	IF TransportItemFound.ID <> '' THEN
		// Test the sorter item against the update item
		IF TransportItemFound.ID = TransportItemInSorter.ID THEN
			// Only update if it is different
			IF TransportItemFound.Destination <> TransportItemInSorter.Destination THEN
				IF .nSortBufferLogEnable.BUFFER_UPDATEDEST THEN
					sMessage := CONCAT(' Item: ', TransportItemInSorter.ID);
					sMessage := CONCAT(sMessage,' Index: ');
					sMessage := CONCAT(sMessage, UDINT_TO_STRING(TransportSorterIndex));
					sMessage := CONCAT(sMessage,' Orig Dest: ');
					sMessage := CONCAT(sMessage, DINT_TO_STRING(TransportItemInSorter.Destination));
					sMessage := CONCAT(sMessage,' Orig DeviceID ');
					sMessage := CONCAT(sMessage, TransportItemInSorter.DeviceID);
					// Write to the Error List
					ADSLOGSTR( msgCtrlMask := ADSLOG_MSGTYPE_HINT OR ADSLOG_MSGTYPE_LOG
						, msgFmtStr := 'Dest Updated After Induct: %s'
						, strArg := sMessage);
				END_IF
				// Update the Destination. If the destination is unavailable, it has been already been set to the default
				TransportItemInSorter.Destination := TransportItemFound.Destination;
				TransportItemInSorter.DeviceID := TransportItemFound.DeviceID;
				TransportItemInSorter.MessageType := TransportItemFound.MessageType;
				TransportItemInSorter.Status := TransportItemFound.Status;
				TransportItemInSorter.ExtStatus := TransportItemFound.ExtStatus;
	
				IF .nSortBufferLogEnable.BUFFER_UPDATEDEST THEN
					sMessage := CONCAT(' Item: ', TransportItemInSorter.ID);
					sMessage := CONCAT(sMessage,' Index: ');
					sMessage := CONCAT(sMessage, UDINT_TO_STRING(TransportSorterIndex));
					sMessage := CONCAT(sMessage,' New Dest: ');
					sMessage := CONCAT(sMessage, DINT_TO_STRING(TransportItemInSorter.Destination));
					sMessage := CONCAT(sMessage,' New DeviceID ');
					sMessage := CONCAT(sMessage, TransportItemInSorter.DeviceID);
					// Write to the Error List
					ADSLOGSTR( msgCtrlMask := ADSLOG_MSGTYPE_HINT OR ADSLOG_MSGTYPE_LOG
						, msgFmtStr := 'Dest Updated After Induct: %s'
						, strArg := sMessage);
				END_IF
			END_IF
			// Make sure that the destination update makes it to the item being inducted into the sorter
			IF st_UpdateItem.Item.ID <> '' THEN
				IF st_UpdateItem.Item.ID = TransportItemFound.ID THEN
					IF st_UpdateItem.Item.Destination <> TransportItemFound.Destination THEN
						IF .nSortBufferLogEnable.BUFFER_UPDATEDEST THEN
							// Log the original destination
							sMessage := CONCAT(' Item: ', st_UpdateItem.Item.ID);
							sMessage := CONCAT(sMessage, ' Pulses: ');
							sMessage := CONCAT(sMessage, UDINT_TO_STRING(st_Sorter.EncoderCounts));
							sMessage := CONCAT(sMessage,' Orig Dest: ');
							sMessage := CONCAT(sMessage, DINT_TO_STRING(st_UpdateItem.Item.Destination));
							// Write to the Error List
							ADSLOGSTR( msgCtrlMask := ADSLOG_MSGTYPE_HINT OR ADSLOG_MSGTYPE_LOG
								, msgFmtStr := 'Induct Dest Changed: %s'
								, strArg := sMessage);
						END_IF
						// Update the Destination
						st_UpdateItem.Item.Destination := TransportItemFound.Destination;
						// Log the new destination
						IF .nSortBufferLogEnable.BUFFER_UPDATEDEST THEN
							sMessage := CONCAT(' Item: ', st_UpdateItem.Item.ID);
							sMessage := CONCAT(sMessage, ' Pulses: ');
							sMessage := CONCAT(sMessage, UDINT_TO_STRING(st_Sorter.EncoderCounts));
							sMessage := CONCAT(sMessage,' New Dest: ');
							sMessage := CONCAT(sMessage, DINT_TO_STRING(st_UpdateItem.Item.Destination));
							// Write to the Error List
							ADSLOGSTR( msgCtrlMask := ADSLOG_MSGTYPE_HINT OR ADSLOG_MSGTYPE_LOG
								, msgFmtStr := 'Induct Dest Changed: %s'
								, strArg := sMessage);
						END_IF
					END_IF
				END_IF
			ELSE
				IF .nSortBufferLogEnable.BUFFER_UPDATEDEST THEN
					sMessage := CONCAT(' Item: ', TransportItemInSorter.ID);
					sMessage := CONCAT(sMessage,' Index: ');
					sMessage := CONCAT(sMessage, UDINT_TO_STRING(TransportSorterIndex));
					sMessage := CONCAT(sMessage,' Orig Dest: ');
					sMessage := CONCAT(sMessage, DINT_TO_STRING(TransportItemInSorter.Destination));
					// Write to the Error List
					ADSLOGSTR( msgCtrlMask := ADSLOG_MSGTYPE_HINT OR ADSLOG_MSGTYPE_LOG
						, msgFmtStr := 'Dest Received After Induct: %s'
						, strArg := sMessage);
				END_IF
				
			END_IF
		END_IF
	END_IF

	// Put the updated record back into the array
	aItems[TransportSorterIndex] := TransportItemInSorter;
	
//==================================================
// 	Done procesing Transport information
//
//	Begin processing Update/Exit information
//==================================================
	
	// For exits, start from the current encoder count and work forward
	ExitSorterIndex := F_CalculateIndex(Offset := UpdateIndexCounter
										, InitialValue := st_Sorter.EncoderCounts
										, BufferSize := ItemsArraySize);

	// Identify the Item we are testing
	ExitItemInSorter := aItems[ExitSorterIndex];

	// Populated ID identifies an item in the sorter
	// Between the two Divert status codes indicates that the item has attempted to divert
	IF ExitItemInSorter.ID <> '' THEN
		// Capture the Item encoder index and the Item at the current index
		//  This represents the first item record for this item
		//  It is captured to log the start index to allow this first record to be updated
		//  when the item is completely diverted
		IF ExitItemFound.Item.ID = '' THEN
			ExitItemFound.Counts := ExitSorterIndex;
			ExitItemFound.Item := ExitItemInSorter;
			IF ExitItemFound.Item.Status = E_StatusCode.Divert_Complete THEN
				ExitComplete := TRUE;
			END_IF
		END_IF
		// When ExitComplete is TRUE, and the ID's match, clear out this Item
		IF ExitComplete THEN
			IF ExitItemInSorter.ID = ExitItemFound.Item.ID THEN
				IF aItems[ExitSorterIndex].ID <> '' THEN
					IF .nSortBufferLogEnable.BUFFER_DUMP THEN
						sMessage := CONCAT(' Item: ', aItems[ExitSorterIndex].ID);
						sMessage := CONCAT(sMessage,' Index: ');
						sMessage := CONCAT(sMessage, UDINT_TO_STRING(ExitSorterIndex));
						sMessage := CONCAT(sMessage,' Item Status: ');
						sMessage := CONCAT(sMessage, DINT_TO_STRING(aItems[ExitSorterIndex].Status));
						sMessage := CONCAT(sMessage,' Item Ext Status: ');
						sMessage := CONCAT(sMessage, DINT_TO_STRING(aItems[ExitSorterIndex].ExtStatus));
						// Write to the Error List
						ADSLOGSTR( msgCtrlMask := ADSLOG_MSGTYPE_HINT OR ADSLOG_MSGTYPE_LOG
							, msgFmtStr := 'Exit Complete Dump Info: %s'
							, strArg := sMessage);
					END_IF
				END_IF
				aItems[ExitSorterIndex] := BlankItem;
			END_IF
		// When ExitComplete is FALSE, test for a diverting/diverted item
		ELSE
			// Detect when this item is in a diverting state
			IF (ExitItemInSorter.Status >= E_StatusCode.Diverting
			   OR ExitItemInSorter.Status <= E_StatusCode.Divert_Success)
			   THEN
			   	ExitInDivert := TRUE;
				(*
					Status value increase from Diverting to Divert_Complete
					Codes to indicate divert disposition are between Diverting and Divert_Detected
					Divert_Full and Diverting are set in FB_DivertDecision/FB_DivertControl
					Divert_Detected, Divert_Success, and Divert_Missed are set in FB_ConfirmCheck
				*)
				ExitDiverting := TRUE;
				IF ExitItemInSorter.Status = E_StatusCode.Divert_Detected THEN
					ExitDetected := TRUE;
				END_IF
				// Once the divert is successful, we are no longer "diverting"
				IF ExitItemInSorter.Status = E_StatusCode.Divert_Success THEN
					ExitSuccess := TRUE;
					ExitDiverting := FALSE;
				END_IF
				(*	
					ExitItemInSorter is the current item being examined
					ExitItemFound.Item is a copy of the Array item at ExitItemFound.Counts
					ExitItemFound.Counts references the Array index of the first record associated with this item
					When a Status/ExtStatus of greater value is detected, the first record Status/ExtStatus is overwritten
					The ExitItemFound.Item.Status/.ExtStatus is also updated
				*)
				IF ExitItemInSorter.Status > aItems[ExitItemFound.Counts].Status THEN
					aItems[ExitItemFound.Counts].Status := ExitItemInSorter.Status;
					ExitItemFound.Item.Status := ExitItemInSorter.Status;
				END_IF
				IF ExitItemInSorter.ExtStatus > aItems[ExitItemFound.Counts].ExtStatus THEN
					aItems[ExitItemFound.Counts].ExtStatus := ExitItemInSorter.ExtStatus;
					ExitItemFound.Item.ExtStatus := ExitItemInSorter.ExtStatus;
				END_IF
			END_IF
			aItems[ExitSorterIndex].Status := ExitItemFound.Item.Status;
		END_IF
	ELSE
		(*
			This path is followed when the ExitItemInSorter.ID is empty, which indicates
			that the array record associated with this index is not occupied

			ExitInDivert, ExitDiverting and ExitSuccess are all set while the .ID is not empty
		*)
		// This item was in a "diverting" state
		IF ExitInDivert THEN
			// This item is not currently diverting
			IF NOT ExitDiverting THEN
				// Only change to a Divert_Success if a Divert_Success was detected
				// Any other status is captured in the ELSE clause of the CASE statement
				IF ExitSuccess THEN
					ExitItemFound.Item.Status := E_StatusCode.Divert_Success;
				END_IF
				ExitItemFound.Item.CapturedInMetrics := TRUE;
				ExitItemFound.Item.MessageType := E_MessageIds.TransportComplete_26;
				fb_UpdateBuffer.AddItem(ExitItemFound.Item);
				aItems[ExitItemFound.Counts].Status := E_StatusCode.Divert_Complete;
			END_IF
		END_IF
		// Clear the last detected Exit item
		ExitItemFound.Item := BlankItem;
		// Reset the Detection booleans
		ExitInDivert := FALSE;
		ExitDiverting := FALSE;
		ExitDetected := FALSE;
		ExitSuccess := FALSE;
		ExitComplete := FALSE;
	END_IF
END_FOR

// If the ID is populated, we didn't find a match to update
IF st_ToUpdate.Item.ID <> '' THEN
	IF .nSortBufferLogEnable.BUFFER_UNASSIGNED THEN
		sMessage := CONCAT(' Item: ', st_ToUpdate.Item.ID);
		// Write to the Error List
		ADSLOGSTR( msgCtrlMask := ADSLOG_MSGTYPE_HINT OR ADSLOG_MSGTYPE_LOG
			, msgFmtStr := 'Item Not Updated: %s'
			, strArg := sMessage);
	END_IF
	st_ToUpdate.Item.Status := E_StatusCode.Assign_NotFound;
	st_ToUpdate.Item.DeviceID := st_Sorter.Config.Name;
	st_ToUpdate.Item.MessageType := E_MessageIds.TransportResponse_25;
	fb_UpDateBuffer.AddItem(st_ItemToAdd := st_ToUpdate.Item);
	st_ToUpdate.Item := BlankItem;
END_IF

END_PROGRAM

// ---- POUs/FunctionBlocks/Sorter/SorterExample.TcPOU
PROGRAM SorterExample
VAR
	nSorterClearIdx				: DINT;
	bSimulate					: BOOL := FALSE;	// Indicates when runing a simulation
	BlankItem					: ST_Item := (ID := ''
												, UniqueID := 0
												, Destination := 0
												, Status := E_StatusCode.No_Status
												, ExtStatus := E_StatusCode.No_Status
												, DeviceID := ''
												, MessageType := E_MessageIds.NoMessage_00);
	
	st_ToInduct					: ST_ItemTemporary;	// This is the next item to be inducted onto the sorter
	st_Inducting				: ST_ItemTemporary;	// This is the next item to be inducted onto the sorter
	st_InductUpdate				: ST_ItemTemporary;	// This is to update an item already being inducted
	{attribute 'OPC.UA.DA' := '1'}
	st_Sorter					: ST_Sorter;
	{attribute 'OPC.UA.DA' := '1'}
	aSorterDiverts 				: ARRAY[DIVERTMIN..NUMBEROFDIVERTS] OF ST_Divert;

	st_SorterEncoder 			: ST_Encoder;
	fb_SorterEncoder 			: FB_ProcessEncoder;
	{attribute 'OPC.UA.DA' := '1'}
	ENC_Raw	AT %I*:	UINT;	// Raw Encoder Value
	tEncoderOK			: TON;
	nLastEncoderCount	: UDINT;

	{attribute 'OPC.UA.DA' := '1'}
	fb_SortMetrics				: FB_Metrics;

	In_DefaultDestination AT %I*	: DINT;	// Input default destination update from Host messaging(MsgControl.RECEIVE)

	fb_CommissionSorterDiverts	: FB_DivertCommission;
	rInductPE					: R_TRIG; 	// Capture the Rising edge of the Induct PE
	fInductPE					: F_TRIG; 	// Capture the Falling edge of the Induct PE

	rDischargePE				: R_TRIG; 	// Capture the Rising edge of the Discharge PE
	fDischargePE				: F_TRIG; 	// Capture the Falling edge of the Discharge PE

	st_TempItem					: ST_ItemTemporary;	// Store temporary Item info until BCR data is received

	DivertToCommission			: UINT := 0;	// Non-zero value will send all items to this divert

	sMessage			: STRING;

	ClearSorterArray	: BOOL;

	FB_DivertLog		: FB_DivertLog;
	
	SorterDischargeItem	: ST_Item;

END_VAR

VAR PERSISTENT
	aSorterItems 				: ARRAY[SORTERENCODERMIN..SORTERENCODERMAX] OF ST_Item;	// Persist the Items to Sort array
	{attribute 'OPC.UA.DA' := '1'}
	st_SorterCfg				: ST_SorterConfig; 	// Persist Sorter configuration
	{attribute 'OPC.UA.DA' := '1'}
	aSorterDivertsCfgs 			: ARRAY[DIVERTMIN..NUMBEROFDIVERTS] OF ST_DivertCfg; 	// Persist Sorter Configuration
END_VAR

VAR CONSTANT
	SORTERMASKSIZE				: UINT := 11;		// Number of bits to mask into the Encoder Count, will define the size of the SORTERENCODERMAX value
	{attribute 'OPC.UA.DA' := '1'}
	NUMBEROFDIVERTS				: DINT := 3;
	DIVERTMIN					: DINT := 1;
	{attribute 'OPC.UA.DA' := '1'}
	SORTERENCODERMAX			: UDINT := ((LREAL_TO_UDINT(EXPT(2,SORTERMASKSIZE)))-1); // Calculated size based on the bitmask 
	{attribute 'OPC.UA.DA' := '1'}
	SORTERENCODERMIN			: UDINT := 0;

END_VAR

// Sorter clear when the system is restarted or downloaded (INIT=TRUE for first scan)
IF (GVL_IO.INIT AND NOT st_SorterCfg.RetainOnRestart) OR ClearSorterArray THEN
	FOR nSorterClearIdx := UDINT_TO_DINT(SORTERENCODERMIN) TO UDINT_TO_DINT(SORTERENCODERMAX) BY 1 DO
		IF nSorterLogEnable.SORTER_DUMP THEN
			IF aSorterItems[nSorterClearIdx].ID <> '' THEN
				IF .nSorterLogEnable.SORTER_DUMP THEN
					sMessage := CONCAT(' Item: ', aSorterItems[nSorterClearIdx].ID);
					sMessage := CONCAT(sMessage,' Index: ');
					sMessage := CONCAT(sMessage, DINT_TO_STRING(nSorterClearIdx));
					// Write to the Error List
					ADSLOGSTR( msgCtrlMask := ADSLOG_MSGTYPE_HINT OR ADSLOG_MSGTYPE_LOG
						, msgFmtStr := 'Array Dump Info: %s'
						, strArg := sMessage);
				END_IF
			END_IF
		END_IF
		aSorterItems[nSorterClearIdx] := BlankItem;
	END_FOR
	ClearSorterArray := FALSE;
END_IF

// Setup and process the Sorter Encoder
st_SorterEncoder.EncoderRawCount := ENC_Raw;
st_SorterEncoder.BitMaskSize := SORTERMASKSIZE;
fb_SorterEncoder(Encoder := st_SorterEncoder, Simulate := bSimulate);

(*
	Initializes the Diverts.  
*)
{warning 'TODO: Fix references to Full and Confirm PE'}
{warning 'TODO: Add Configuration for all Diverts'}
aSorterDiverts[1].Config := aSorterDivertsCfgs[1];
aSorterDiverts[1].FullPE := TRUE;
aSorterDiverts[1].ConfirmPE := TRUE;

fb_CommissionSorterDiverts(
			//InductTrigger := Photoeyes.PE_22441.Out,
			ReferenceValue := st_SorterEncoder.CurrentCount, 
			//DischargeTrigger := Photoeyes.PE_23121.Out_OffFltrd,
			TestTime := T#10S, Diverts := aSorterDiverts);

// Provide a "hard-coded" default destination.
IF st_SorterCfg.DefaultDestination <= 0 THEN
	st_SorterCfg.DefaultDestination := 1;
END_IF						

// Name of the sorter equipment
//st_SorterCfg.Name := Conveyors.cfgP8005Label;
st_SorterCfg.DivertCount := NUMBEROFDIVERTS;
IF DivertToCommission > 0 THEN
	st_SorterCfg.DefaultDestination := DivertToCommission;
END_IF
st_Sorter.EncoderCounts := st_SorterEncoder.CurrentCount;
//st_Sorter.InductPE := PhotoEyes.PE_22441.Out_OnFltrd;
//st_Sorter.DischargePE := Photoeyes.PE_23081.Out_OnFltrd;

// Test the Encoder
//tEncoderOK.IN := (Conveyors.P8005_VFD.IsRunning AND (st_Sorter.EncoderCounts = nLastEncoderCount));
tEncoderOK(PT:=T#1S);

// OK when Q is not on, but the alarm is reversed
//GVL_IO.ENC_11321_OK := tEncoderOK.Q;

// Publish the sorter name
//GVL_IO.SorterName := st_SorterCfg.Name;

// Sorter
(*
	ProcessBuffers processes all associated buffers (Sorter/Divert/Arrival/Transport/Update)
	Items arriving at the sorter are detected and processed in this function block then deliverd to the SorterProgram
	Items inducted into sorter produce TransportResponse messages in this function block
	Items diverted off the sorter produce TransportComplete messages in this function block
*)
ProcessBuffers(st_NextToInduct := st_ToInduct
				, st_TempInductItem := st_TempItem
				, st_UpdateItem := st_Inducting
				, st_Sorter := st_Sorter
				, aDiverts := aSorterDiverts
				, aItems := aSorterItems
				, DivertToCommission := DivertToCommission
				, ItemsArrayMax := SORTERENCODERMAX
				, ItemsArrayMin := SORTERENCODERMIN);

// Capture rising and falling edge Triggers of the configured Sorter PE (Induct/Discharge)
rInductPE(CLK:= st_Sorter.InductPE, Q =>);
fInductPE(CLK:= st_Sorter.InductPE, Q =>);
rDischargePE(CLK:= st_Sorter.DischargePE, Q =>);
fDischargePE(CLK:= st_Sorter.DischargePE, Q =>);

// Prepare a dummy record for items that arrive before BCR data is received
// On the rising edge of the Induct PE
IF rInductPE.Q THEN
	IF .nSorterLogEnable.SORTER_INDUCT_PE THEN
		// Write to the Error List
		ADSLOGSTR( msgCtrlMask := ADSLOG_MSGTYPE_HINT OR ADSLOG_MSGTYPE_LOG
			, msgFmtStr := 'Induct PE Blocked : %s'
			, strArg := BOOL_TO_STRING(st_Sorter.InductPE)); 
	END_IF
	// Test for a UniqueID, which indicates that a Barcode has been received
	IF st_ToInduct.Item.UniqueID = 0 THEN
		// Capture and create relevant info
		st_TempItem.Counts := st_Sorter.EncoderCounts;
		st_TempItem.Item.UniqueID :=  UDINT_TO_DINT(st_Sorter.EncoderCounts);
		st_TempItem.Item.ID :=  CONCAT('T-', UDINT_TO_STRING(st_Sorter.EncoderCounts));
		st_TempItem.Item.Destination := st_SorterCfg.DefaultDestination;
		st_TempItem.Item.Status := E_StatusCode.UnidentifiedItem;
		IF .nSorterLogEnable.SORTER_TEMPID THEN
			ADSLOGSTR( msgCtrlMask := ADSLOG_MSGTYPE_HINT OR ADSLOG_MSGTYPE_LOG
				, msgFmtStr := 'Temp ID Assigned : %s'
				, strArg := st_TempItem.Item.ID);
		END_IF
	END_IF	
END_IF

// Clear the dummy record when the PE clears
// Items can only be inducted when the BCR info is received before or while the induct PE is blocked
IF fInductPE.Q THEN
	IF .nSorterLogEnable.SORTER_INDUCT_PE THEN
		// Write to the Error List
		ADSLOGSTR( msgCtrlMask := ADSLOG_MSGTYPE_HINT OR ADSLOG_MSGTYPE_LOG
			, msgFmtStr := 'Induct PE Blocked : %s'
			, strArg := BOOL_TO_STRING(st_Sorter.InductPE));
	END_IF
	// Clear the record
	st_TempItem.Counts := 0;
	st_TempItem.Item :=  BlankItem;
END_IF

(*
	SorterProgram is a separate Program
	Config portion of the st_sorter is separate to allow it be be persistent.
*)
st_sorter.Config := st_sorterCfg;
SorterProgram(st_Sorter := st_Sorter
		, In_ItemToInduct := st_ToInduct.Item
		, In_InductingItem := st_Inducting.Item
		, aItems := aSorterItems
		, aDiverts := aSorterDiverts
		, st_tempItem := st_TempItem
		, ItemsArrayMax := SORTERENCODERMAX
		, ItemsArrayMin := SORTERENCODERMIN
		, DivertArrayMax := DIVERTMIN
		, DivertArrayMin := NUMBEROFDIVERTS
		, st_DischargeItem => SorterDischargeItem);

// Log the diverts
FB_DivertLog(DivertArray := aSorterDiverts,
				DivertLogEnable := .nDivertLogEnable,
				EncoderCounts := st_SorterEncoder.CurrentCount);

END_PROGRAM

// ---- POUs/FunctionBlocks/Sorter/Functions/FB_FindDestination.TcPOU
FUNCTION_BLOCK FB_FindDestination
VAR_IN_OUT
	RoundRobin		:	ST_RoundRobin;
	aDiverts		:	ARRAY[*] OF ST_Divert;
	DestinationID	:	DINT;
END_VAR
VAR_INPUT
	SorterLogEnable	:	UDINT;
END_VAR
VAR_OUTPUT
	DestinationIndex	:	DINT;
	DestinationState	:	DINT;
END_VAR
VAR
	DivertArrayMin		:	DINT;
	DivertArrayMax		:	DINT;
	Last_Enabled	:	UINT;
	IndexCheck		:	DINT;
	sMessage		:	STRING;
END_VAR

// Get the upper and lower bounds of the divert array
DivertArrayMin := LOWER_BOUND(aDiverts,1);
DivertArrayMax := UPPER_BOUND(aDiverts,1);

//When a response is received, find the designated Destination
IF DestinationID >= 0 THEN
	IF SorterLogEnable.SORTER_DESTINATION_LU THEN
		sMessage := CONCAT(' Destination: ', DINT_TO_STRING(DestinationID));
		// Write to the Error List
		ADSLOGSTR( msgCtrlMask := ADSLOG_MSGTYPE_HINT OR ADSLOG_MSGTYPE_LOG
			, msgFmtStr := 'Lookup: %s'
			, strArg := sMessage);
	END_IF
	// Check to see if the Destination is defined as a round-robin destination for this sorter
	IF DestinationID = RoundRobin.Destination THEN
		// Test to see if the last enabled round robin destinations are still enabled
		// If they are different, restart the round-robin assignment to accommodate differences 
		IF RoundRobin.Enabled = Last_Enabled THEN
			// Test to see if the round robin assignments have all been met
			// If they have, clear and start over
			IF RoundRobin.Available = RoundRobin.Sent THEN
				RoundRobin.Sent := 0;
			END_IF
		ELSE
			// Capture the new enabled round-robin destinations
			// Restart the round robin assignments
			Last_Enabled := RoundRobin.Enabled;
			RoundRobin.Sent := 0;
		END_IF
		FOR IndexCheck := 0 TO 15 DO
			IF (
			   ((RoundRobin.Enabled AND LREAL_TO_UINT(EXPT(2,IndexCheck))) > 0) 
			   AND ((RoundRobin.Available AND LREAL_TO_UINT(EXPT(2,IndexCheck))) > 0)
			   AND NOT ((RoundRobin.Sent AND LREAL_TO_UINT(EXPT(2,IndexCheck))) > 0))
			   THEN
				RoundRobin.Sent := LREAL_TO_UINT(EXPT(2,IndexCheck)) OR RoundRobin.Sent;
				IF RoundRobin.aDestinations[IndexCheck] >= DivertArrayMin
				   AND RoundRobin.aDestinations[IndexCheck] <= DivertArrayMax
				   THEN
					DestinationIndex := RoundRobin.aDestinations[IndexCheck];
					DestinationID := aDiverts[DestinationIndex].Config.Number;
				ELSE
					DestinationIndex := DivertArrayMax;
				END_IF
				DestinationState := 0;
				EXIT;
			END_IF
		END_FOR
		IF SorterLogEnable.SORTER_DESTINATION_LU THEN
			sMessage := DINT_TO_STRING(DestinationIndex);
			sMessage := CONCAT(' Dest ID: ', DINT_TO_STRING(DestinationID));
			// Write to the Error List
			ADSLOGSTR( msgCtrlMask := ADSLOG_MSGTYPE_HINT OR ADSLOG_MSGTYPE_LOG
				, msgFmtStr := 'RoundRobin Dest: %s'
				, strArg := sMessage);
		END_IF
	ELSE
		DestinationIndex := DivertArrayMax;
		FOR IndexCheck := DivertArrayMin TO DivertArrayMax  DO
			IF aDiverts[IndexCheck].Config.Number = DestinationID THEN
				DestinationIndex := IndexCheck;
				DestinationState := 0;
				EXIT;
			END_IF
		END_FOR
		IF SorterLogEnable.SORTER_DESTINATION_LU THEN
			sMessage := DINT_TO_STRING(DestinationIndex);
			sMessage := CONCAT(' Dest ID: ', DINT_TO_STRING(DestinationID));
			// Write to the Error List
			ADSLOGSTR( msgCtrlMask := ADSLOG_MSGTYPE_HINT OR ADSLOG_MSGTYPE_LOG
				, msgFmtStr := 'Lookup Dest: %s'
				, strArg := sMessage);
		END_IF
	END_IF
END_IF

END_FUNCTION_BLOCK

// ---- POUs/Sorter_P6040.TcPOU
PROGRAM Sorter_P6040

VAR_IN_OUT
	In_ItemToInduct					: ST_Item;
	In_InductingItem				: ST_Item;
	st_tempItem						: ST_ItemTemporary;	// Temporary record used when barcode not yet received
	st_Sorter						: ST_Sorter;
	aDiverts						: ARRAY[Sorter.DIVERTMIN..Sorter.NUMBEROFDIVERTS] OF ST_DIVERT;
	aItems 							: ARRAY[Sorter.SORTERENCODERMIN..Sorter.SORTERENCODERMAX] OF ST_Item;
END_VAR

VAR_INPUT
	ItemsArrayMax		: UDINT;
	ItemsArrayMin		: UDINT;
	DivertArrayMax		: DINT;
	DivertArrayMin		: DINT;
END_VAR

VAR_OUTPUT
	st_DischargeItem	:	ST_Item;
END_VAR
VAR
	// Sorter Diagnostics
	aSorterDiagLog		: ST_ItemLogBuffer;
	fbSorterDiagLog		: FB_ItemLogBuffer;

	//Logging Variables
	UpdateSorterLog : FB_UpdateLog;
	
	//Induct Variables
	testEncoderCount		: UDINT;
	exitEncoderCount		: UDINT;
	lastCompareCount		: UDINT;
	updatingEncoderCount	: UDINT;

	tailendcount		: DINT := 0;
	inductindex 		: DINT;
	
	//Divert Variables
	fb_DivertDecision 		: FB_DivertDecision;
	fb_DivertFullMonitor  	: FB_DivertFullMonitor;
	DivertIndex				: DINT;
	Divertoffset			: INT;
	nTestItemIndex			: UDINT;
	Output2ItemIndex		: UDINT;

	// Confirm Check variables
	fb_ConfirmCheck 		: ARRAY[Sorter.DIVERTMIN..Sorter.NUMBEROFDIVERTS] OF FB_ConfirmCheck;
	st_ConfirmItem 			: ARRAY[Sorter.DIVERTMIN..Sorter.NUMBEROFDIVERTS] OF ST_Item;
	nConfirmItemIndex 		: UDINT;
	
	workingItem			: ST_Item;	// Actual item to induct

	LastItemInducted 	: STRING;
	nIndexToClear		: UDINT;	// Clear Item Array at this index
	nItemArraySize		: UDINT;

	rInductPE			: R_TRIG; 	// Capture the Rising edge of the Induct PE
	fInductPE			: F_TRIG; 	// Capture the Falling edge of the Induct PE
	sMessage			: STRING;

	st_DisplayItem		:st_Item;
	
	LogSorterDump: BOOL := FALSE;
END_VAR

// Initialize FB_ItemExtBuffer
fbSorterDiagLog(st_BufferData := aSorterDiagLog);

(*
// Test visu variables	
inductPE := SorterInductPE;
ItemsOut := Items;
ArrivalOut := ArrivalBuffer;
// End test variables
*)
(*
	Capture the Upper/Lower bound of relevant IO_OUT arrays for looping purposes
	ItemsArrayMax/Min for the sorter array slot count
*)
// Size is Max - Min + 1 to capture both extremes
nItemArraySize := ItemsArrayMax - ItemsArrayMin + 1;

FOR divertIndex := DivertArrayMin TO DivertArrayMax DO
	fb_DivertFullMonitor(Divert := aDiverts[divertIndex]);
END_FOR

(*
	Detect barcode receipt after item is already in Item array
	the tempItem is reset when the induct PE is cleared
	The tempItem is populated when the induct PE is blocked and there
	is not an associated barcode waiting to be inducted
*)
IF st_tempItem.Item.ID <> '' THEN
	// Test the IN_ItemToInduct.ID for a value
	// This record will be cleared as soon as it reaches the sorter loop
	IF In_ItemToInduct.ID <> '' THEN
		// The tempItem is overwritten with the IN_ItemToInduct after it is updated
		// But the starting encoder count is not changed so the same items can be updated
		// if the destination update is received while the item is still being inducted
		IF In_ItemToInduct.ID <> st_tempItem.Item.ID THEN 
			// Set the starting count for the testing/updating process
			// The testEncodeCount is incremented upon start, so we start -1 of the encoder count for the item
			testEncoderCount := f_CalculateIndex(Offset := -1, InitialValue:= st_tempItem.Counts, BufferSize := nItemArraySize);
			// Clear the length and start over
			In_ItemToInduct.Length := 0;
			st_tempItem.Item := In_ItemToInduct;
		END_IF 
		// Test for a change of destination after the barcode data has been received
		IF In_ItemToInduct.Destination <> st_tempItem.Item.Destination THEN 
			// Set the starting count for the testing/updating process
			// The testEncodeCount is incremented upon start, so we start -1 of the encoder count for the item
			testEncoderCount := f_CalculateIndex(Offset := -1, InitialValue:= st_tempItem.Counts, BufferSize := nItemArraySize);
			// Clear the length and start over
			In_ItemToInduct.Length := 0;
			// Copy the IN_ItemToInduct to prevent running this until something else in the record changes
			st_tempItem.Item := IN_ItemToInduct;
		END_IF
	END_IF 
END_IF


// Test for the rising edge of the induct PE
// Use this rising edge to log the IN_ItemToInduct record
rInductPE(CLK:= st_Sorter.InductPE, Q =>);

IF rInductPE.Q THEN
	IF .nSorterLogEnable.SORTER_INDUCT THEN
		sMessage := CONCAT(' Item: ', In_ItemToInduct.ID);
		sMessage := CONCAT(sMessage, ' Pulses: ');
		sMessage := CONCAT(sMessage, UDINT_TO_STRING(st_Sorter.EncoderCounts));
		// Write to the Error List
		ADSLOGSTR( msgCtrlMask := ADSLOG_MSGTYPE_HINT OR ADSLOG_MSGTYPE_LOG
			, msgFmtStr := 'Induct Info: %s'
			, strArg := sMessage);
	END_IF
END_IF
// Test for the falling edge of the induct PE
// Use this falling edge to clear the IN_ItemToInduct record
fInductPE(CLK:= st_Sorter.InductPE, Q =>);

IF fInductPE.Q THEN
	IF .nSorterLogEnable.SORTER_INDUCT THEN
		sMessage := CONCAT(' Item: ', In_ItemToInduct.ID);
		sMessage := CONCAT(sMessage,' Pulses: ');
		sMessage := CONCAT(sMEssage, UDINT_TO_STRING(st_Sorter.EncoderCounts));
		// Write to the Error List
		ADSLOGSTR( msgCtrlMask := ADSLOG_MSGTYPE_HINT OR ADSLOG_MSGTYPE_LOG
			, msgFmtStr := 'Cleared Induct Info: %s'
			, strArg := sMessage);
	END_IF
	// Clear the record
	In_InductingItem :=  BlankItem;
END_IF

// Process every array index between the current index and the last processed index
WHILE st_Sorter.EncoderCounts <> testEncoderCount DO

	// Capture the lastEncoderCount before changing it for comparison of last inducted items
	lastCompareCount := testEncoderCount;

	// Increment the testEncoderCount
	// The testEncoderCount variable will be used throughout the processing to ensure
	//	that all array elements are processed
	testEncoderCount := f_CalculateIndex(Offset := 1, InitialValue:= testEncoderCount, BufferSize := nItemArraySize);
	IF st_Sorter.InductPE THEN
	  	IF (In_ItemToInduct.ID <> '') THEN
			In_InductingItem := In_ItemToInduct;
			In_ItemToInduct := BlankItem;
			IF .nSorterLogEnable.SORTER_INDUCT_PE THEN
				sMessage := CONCAT(' Item: ', In_InductingItem.ID);
				sMessage := CONCAT(sMessage,' Pulses: ');
				sMessage := CONCAT(sMessage, UDINT_TO_STRING(st_Sorter.EncoderCounts));
				sMessage := CONCAT(sMessage,' Dest: ');
				sMessage := CONCAT(sMessage, DINT_TO_STRING(In_InductingItem.Destination));
				// Write to the Error List
				ADSLOGSTR( msgCtrlMask := ADSLOG_MSGTYPE_HINT OR ADSLOG_MSGTYPE_LOG
					, msgFmtStr := 'Inducting Info: %s'
					, strArg := sMessage);
			END_IF
		END_IF
	  	IF (In_InductingItem.ID <> '') THEN
			LastItemInducted := In_InductingItem.ID;
			IF aItems[testEncoderCount].ID <> '' THEN
				IF aItems[testEncoderCount].Status >= E_StatusCode.Diverting AND aItems[testEncoderCount].Status <= E_StatusCode.Divert_UnknownError THEN
					aItems[testEncoderCount].Status := E_StatusCode.Divert_UnknownError;
				END_IF
				UpdateSorterLog(Status := aItems[testEncoderCount].Status, ItemID := aItems[testEncoderCount].UniqueID);
			END_IF
		
			// Set the Item status
			In_InductingItem.Status := E_StatusCode.In_Sorter;

			// Check for destination full on the first pass, then ignore it.
		IF In_InductingItem.Length = 0 THEN
				IF aDiverts[In_InductingItem.DestinationIdx].Full THEN
					IF st_Sorter.Config.RecircUsed THEN
						In_InductingItem.Destination := st_Sorter.Config.RecircDestination;
						In_InductingItem.DestinationIdx := st_Sorter.Config.RecircDestIdx;
						In_InductingItem.ExtStatus := E_StatusCode.Divert_Recirculated;
					ELSE
						In_InductingItem.Destination := st_Sorter.Config.DefaultDestination;
						In_InductingItem.DestinationIdx := st_Sorter.Config.DefaultDestIdx;
						In_InductingItem.ExtStatus := E_StatusCode.Divert_Full;
					END_IF
				END_IF
			END_IF 
			// Clear the extend counter
			tailendcount := 0;

			// Copy the ItemToInduct to the WorkingItem that will be inducted
			workingItem := In_InductingItem;
			// Increment the Length on the ItemToInduct record, then it will be added to the array
			//  and the length will increment
			In_InductingItem.Length := In_InductingItem.Length +  1;
			// Determined by UniqueID = 0
		ELSE //If the item makes it to the sorter, but is not identified, induct the item with tempItem.Item
			LastItemInducted := 'UNKNOWN';
			(*UpdateSorterLog(Status := E_StatusCode.UnidentifiedItem, ItemID := st_tempItem.Item.UniqueID);*)

			// Process this the first time
			IF st_tempItem.Item.Length = 0 THEN
				IF aDiverts[st_Sorter.Config.DefaultDestIdx].Full THEN
					IF st_Sorter.Config.RecircUsed THEN
						st_tempItem.Item.Destination := st_Sorter.Config.RecircDestination;
						st_tempItem.Item.DestinationIdx := st_Sorter.Config.RecircDestIdx;
						st_tempItem.Item.ExtStatus := E_StatusCode.Divert_Recirculated;
					ELSE
						st_tempItem.Item.Destination := st_Sorter.Config.DefaultDestination;
						st_tempItem.Item.DestinationIdx := st_Sorter.Config.DefaultDestIdx;
						st_tempItem.Item.ExtStatus := E_StatusCode.Divert_Full;
					END_IF
				ELSE
					st_tempItem.Item.Destination := st_Sorter.Config.DefaultDestination;
					st_tempItem.Item.DestinationIdx := st_Sorter.Config.DefaultDestIdx;
				END_IF		
			END_IF
			// Copy the tempItem.Item to the WorkingItem that will be inducted
			workingItem := st_tempItem.Item;
			// Increment the Length on the ItemToInduct record, then it will be added to the array
			//  and the length will increment
			st_tempItem.Item.Length := st_tempItem.Item.Length +  1;
		END_IF

		// Induct everything
		aItems[testEncoderCount] := workingItem;
		fbSorterDiagLog.AddItem(workingItem);
	// Follow this path when the induct photo-eye is cleared
	ELSE
		// Extend the end of the item by a set amount, or to a mimimum length
		// Test to verify that the Item index is clear, and we are still extending the length of the item
		IF aItems[lastCompareCount].ID <> '' THEN
			IF tailendcount < st_Sorter.Config.TailEndLength AND st_Sorter.Config.TailEndLength > 0 THEN
				aItems[testEncoderCount] := aItems[lastCompareCount]; 
				fbSorterDiagLog.AddItem(aItems[lastCompareCount]);
				aItems[testEncoderCount].Length := aItems[testEncoderCount].Length + 1;
				tailendcount := tailendcount + 1;
			END_IF
			IF aItems[lastCompareCount].Length < st_Sorter.Config.MinimumLength AND st_Sorter.Config.MinimumLength > 0 THEN
				aItems[testEncoderCount] := aItems[lastCompareCount]; 
				fbSorterDiagLog.AddItem(aItems[lastCompareCount]);
				aItems[testEncoderCount].Length := aItems[testEncoderCount].Length + 1;
			END_IF
		END_IF
	END_IF
END_WHILE

// Process every array index between the current index and the last processed exit index
WHILE st_Sorter.EncoderCounts <> exitEncoderCount DO

	// Increment the exitEncoderCount
	// The exitEncoderCount variable will be used throughout the processing to ensure
	//	that all array elements are processed
	exitEncoderCount := f_CalculateIndex(Offset := 1, InitialValue:= exitEncoderCount, BufferSize := nItemArraySize);
	// Process the diverts relative to the current encoder count
	FOR divertIndex := DivertArrayMin TO DivertArrayMax DO
		// Get the distance to each divert, distance is the number of pulses to actuation
		Divertoffset := aDiverts[divertIndex].Config.Distance;
		// Calculate the index of the item to test for a divert
		// Subtract the offset from the current encoder count (exitEncoderCount)
		// As the encoder count increases, the current index pointer advances
		// Subtracting looks backwards into the sorter item array to test for items at the diverts
		//	distance that should be diverted
		nTestItemIndex := F_CalculateIndex(initialvalue := exitEncoderCount
										, offset := -(Divertoffset)
										, BufferSize := (ItemsArrayMax + 1));	
		//Setup Out2Item for energizing 2nd divert output
		Output2ItemIndex := F_CalculateIndex(initialvalue := exitEncoderCount
										, offset := -(Divertoffset + UINT_TO_INT(st_Sorter.Config.Output2Offset))
										, BufferSize := (ItemsArrayMax + 1));	
		// Log Diverts
		IF aItems[nTestItemIndex].DestinationIdx = divertIndex THEN
			IF .nSorterLogEnable.SORTER_DIVERTS THEN
				sMessage := CONCAT(' Item: ', aItems[nTestItemIndex].ID);
				sMessage := CONCAT(sMessage,' Index: ');
				sMessage := CONCAT(sMessage, UDINT_TO_STRING(nTestItemIndex));
				sMessage := CONCAT(sMessage,' Dest: ');
				sMessage := CONCAT(sMessage, DINT_TO_STRING(aItems[nTestItemIndex].Destination));
				sMessage := CONCAT(sMessage,' DestIdx: ');
				sMessage := CONCAT(sMessage, DINT_TO_STRING(aItems[nTestItemIndex].DestinationIdx));
				sMessage := CONCAT(sMessage,' Divert Status: ');
				sMessage := CONCAT(sMessage, DINT_TO_STRING(aDiverts[DivertIndex].Status));
				sMessage := CONCAT(sMessage,' Item Status: ');
				sMessage := CONCAT(sMessage, DINT_TO_STRING(aItems[nTestItemIndex].Status));
				// Write to the Error List
				ADSLOGSTR( msgCtrlMask := ADSLOG_MSGTYPE_HINT OR ADSLOG_MSGTYPE_LOG
					, msgFmtStr := 'Item at Divert Index: %s'
					, strArg := sMessage);
			END_IF
		END_IF
		fb_DivertDecision( bLog := .nDivertLogEnable.DIVERT_DECISION 
					 , Output1Item		:= aItems[nTestItemIndex]
					 , Output2Item		:= aItems[Output2ItemIndex]
					 , Divert 			:= aDiverts[DivertIndex]
					 , DivertIndex		:= DivertIndex
					 );
		// Calculate the distance to the confirm PE to test for a successful divert
		nConfirmItemIndex := F_CalculateIndex(initialvalue := exitEncoderCount
										, offset := -(Divertoffset + aDiverts[divertIndex].Config.ConfirmDist)
										, BufferSize := (ItemsArrayMax + 1));
		// Log Confirms
		IF aItems[nConfirmItemIndex].Status = E_StatusCode.Diverting AND aItems[nConfirmItemIndex].UniqueID <> 0 THEN
			IF .nSorterLogEnable.SORTER_CONFIRMS THEN
				sMessage := CONCAT(' Item: ', aItems[nConfirmItemIndex].ID);
				sMessage := CONCAT(sMessage,' Index: ');
				sMessage := CONCAT(sMessage, UDINT_TO_STRING(nConfirmItemIndex));
				sMessage := CONCAT(sMessage,' Dest: ');
				sMessage := CONCAT(sMessage, DINT_TO_STRING(aItems[nConfirmItemIndex].Destination));
				sMessage := CONCAT(sMessage,' DestIdx: ');
				sMessage := CONCAT(sMessage, DINT_TO_STRING(aItems[nConfirmItemIndex].DestinationIdx));
				sMessage := CONCAT(sMessage,' Divert Status: ');
				sMessage := CONCAT(sMessage, DINT_TO_STRING(aDiverts[DivertIndex].Status));
				sMessage := CONCAT(sMessage,' Item Status: ');
				sMessage := CONCAT(sMessage, DINT_TO_STRING(aItems[nTestItemIndex].Status));
				// Write to the Error List
				ADSLOGSTR( msgCtrlMask := ADSLOG_MSGTYPE_HINT OR ADSLOG_MSGTYPE_LOG
					, msgFmtStr := 'Item at Confirm Index: %s'
					, strArg := sMessage);
			END_IF
		END_IF
		fb_ConfirmCheck[divertIndex] ( bLog := .nDivertLogEnable.DIVERT_DECISION 
					 , ConfirmItem		:= aItems[nConfirmItemIndex]
					 , ConfirmPE 		:= aDiverts[DivertIndex].ConfirmPE
					 , DivertIndex		:= DivertIndex
					 , bIsDischarge		:= aDiverts[DivertIndex].Config.IsDischarge
					 , DetectedItem => st_ConfirmItem[DivertIndex]
					 );
	END_FOR
	
	// Capture the last item discharged by this sorter section
	IF st_ConfirmItem[DivertArrayMax].ID <> '' THEN
		st_DischargeItem := st_ConfirmItem[DivertArrayMax];
	END_IF

	// Clear the Item array ahead of the current encoder count
	nIndexToClear := f_CalculateIndex(Offset := 40, InitialValue:= exitEncoderCount, BufferSize := nItemArraySize);
	IF aItems[nIndexToClear].ID <> '' THEN
		IF .nSorterLogEnable.SORTER_DUMP THEN
			sMessage := CONCAT(' Item: ', aItems[nIndexToClear].ID);
			sMessage := CONCAT(sMessage,' Index: ');
			sMessage := CONCAT(sMessage, UDINT_TO_STRING(nIndexToClear));
			sMessage := CONCAT(sMessage,' Item Status: ');
			sMessage := CONCAT(sMessage, DINT_TO_STRING(aItems[nIndexToClear].Status));
			// Write to the Error List
			ADSLOGSTR( msgCtrlMask := ADSLOG_MSGTYPE_HINT OR ADSLOG_MSGTYPE_LOG
				, msgFmtStr := 'Clear Ahead Dump Info: %s'
				, strArg := sMessage);
		END_IF
	END_IF
	aItems[nIndexToClear] := BlankItem;

END_WHILE

END_PROGRAM

// ---- POUs/FunctionBlocks/Divert/Functions/FB_DivertDecision.TcPOU
FUNCTION_BLOCK FB_DivertDecision
VAR_IN_OUT
	Output1Item 		: ST_Item;
	Output2Item			: ST_Item;
	Divert 				: ST_Divert;
END_VAR

VAR_INPUT
	DivertIndex 		: DINT;
	bLog				: BOOL;
END_VAR

VAR
	DivertController	: FB_DivertControl;
	Output1Activate 	: BOOL := 0;
	Output2Activate 	: BOOL := 0;	
	UpdateLog 			: FB_UpdateLog;
	LastDest 			: DINT;	
	aDivertLog			: ST_ItemLogBuffer;
	fbDivertLog			: FB_ItemLogBuffer;
	ItemToLog			: ST_Item;
	sMessage			: STRING;
END_VAR

fbDivertLog(st_BufferData := aDivertLog);

//Divert this item if this divert is this item's intended destination
IF DivertIndex = Output1Item.DestinationIdx THEN
	// Check this only once, then set the Status accordingly
	IF Divert.Status = E_StatusCode.Divert_Idle THEN
		IF Divert.Full THEN
			Divert.Status := E_StatusCode.Divert_Full;
		else
			Divert.Status := E_StatusCode.Diverting;
		END_IF
		IF bLog THEN
			sMessage := CONCAT(' Item: ', Output1Item.ID);
			sMessage := CONCAT(sMessage,' Dest: ');
			sMessage := CONCAT(sMessage, DINT_TO_STRING(Output1Item.Destination));
			sMessage := CONCAT(sMessage,' Dest: ');
			sMessage := CONCAT(sMessage, DINT_TO_STRING(Output1Item.DestinationIdx));
			sMessage := CONCAT(sMessage,' Status: ');
			sMessage := CONCAT(sMessage, DINT_TO_STRING(Divert.Status));
			// Write to the Error List
			ADSLOGSTR( msgCtrlMask := ADSLOG_MSGTYPE_HINT OR ADSLOG_MSGTYPE_LOG
				, msgFmtStr := 'Divert Initiated: %s'
				, strArg := sMessage);
		END_IF
	END_IF;
	IF Divert.Status = E_StatusCode.Diverting THEN
		Output1Activate := 1;
		Divert.Item := Output1Item;
		//Energize Output2 after SorterCode.CFG_Output2Offset has passed 
		IF DivertIndex = Output2Item.DestinationIdx THEN
			Output2Activate := 1;
		END_IF
		DivertController( Output1Activate	:= Output1Activate
				, Output2Activate	:= Output2Activate
				, Output1Item		:= Output1Item
				, Output2Item		:= Output2Item
				, Divert			:= Divert
				);		
	ELSIF Divert.Status = E_StatusCode.Divert_Full THEN
		Output1Item.ExtStatus := E_StatusCode.Divert_Full;
	END_IF				
//	Output1Item.Status := Divert.Status; 
	ItemToLog := Output1Item;
	ItemToLog.Length := DivertIndex;
	fbDivertLog.AddItem(ItemToLog);
ELSE
	//Turn off output if dest does not equal divert index
	Output1Activate := 0;
	//Keep Output2 energized for SorterCode.CFG_Output2Offset distance
	IF DivertIndex <> Output2Item.DestinationIdx THEN
		// Set and Idle status for the divert
		Divert.Status := E_StatusCode.Divert_Idle;
		Output2Activate := 0;
	ELSE
		Output2Activate := 1;	
	END_IF	

	DivertController( Output1Activate	:= Output1Activate
				, Output2Activate	:= Output2Activate
				, Output1Item		:= Output1Item
				, Output2Item		:= Output2Item
				, Divert			:= Divert
				);
END_IF

END_FUNCTION_BLOCK

// ---- POUs/MsgControl.TcPOU
PROGRAM MsgControl
VAR_INPUT
	TransmitEnable 				: BOOL;
	nConnectionIndex			: UDINT := 1;
END_VAR
VAR
	MsgID						: DINT;			// TCP/IP Message ID as per Communication protocol defined in FA 
	DeviceID					: STRING(5);	// TCP/IP Device ID as per Communication protocol defined in FA 
	BarCode						: STRING(20);	// TCP/IP Load ID (Bar Code) as per Communication protocol defined in FA
	BarCodeNoSpace				: STRING(20);	// TCP/IP Load ID (Bar Code) as per Communication protocol defined in FA stripped of spaces  
	Destination					: DINT;			// TCP/IP Destination as per Communication protocol defined in FA
	DefDestination				: DINT;			// TCP/IP Default Destination as per Communication protocol defined in FA
	Status						: BYTE;				// 
	Msg_EquipStatArry			: ARRAY[1..7] OF ST_Msg_EquipStat;
	nSystemStatusIndex 			: DINT; 	// Index used for Processing the system status array
	nTempOperState 				: DINT;	//Capture the Temporary Operating State of the Equipment for comparison
	nEquipStatusIndex			: DINT;	//Index used for adding items to the MSG_EquipStatArray
	StrStartPos					: INT;
	StrEndPos					: INT;
	MsgString					: STRING(55);
	RawMsgArray					: ARRAY[1..10] OF T_MaxString;	// Capture the last Raw messages for troubleshooting
	RawMsgLenArray				: ARRAY[1..10] OF INT;			// Capture the last  Raw message lengths for troubleshooting
	RawMsgStartPosArray			: ARRAY[1..10] OF INT;			// Capture the last  Raw message start positions for troubleshooting
	RawMsgEndPosArray			: ARRAY[1..10] OF INT;			// Capture the last  Raw message end positions for troubleshooting
	MsgArray					: ARRAY[1..10] OF STRING(55);		// Capture the last 10 messages that have been stripped from the starting character  for troubleshooting
	Blank_Msg_ConveyorStatArry	: ARRAY [1..7] OF ST_Msg_EquipStat := [7((Status := 99))];

	i 							: INT;
	j							: INT;
	
	RxCounter_Old				: UDINT;
	TxCounter_Old				: UDINT;
	TransmitMsgBuffer			: ARRAY [1..TransmitMsgBuffer_Size] OF STRING(55);	// Buffer to hold transmit messages
	TransmitMsgBuffer_Index		: INT :=	1;		// Index to the Buffer
	TransmitMsgStatus			: INT;			
	SendingMsg_Index			: INT :=	1;		// Index to send message
	
	ItemTransport				: ST_Item;		// Output Item Update with destination from ARUP Host (Send to Sorter PLC)

	ReadBCRID_S6040_01_Old			: UDINT;		// Bar Code watch variable
	ReadBCRID_S7004_01_Old			: UDINT;		// Bar Code watch variable

		
	TransmittedArray			: ARRAY[0..10] OF STRING(55);
	x							: DINT;
	y							: INT;
	
	SpacePosition				: INT;
	
	fb_CheckStopRegister		: FB_ManageCodes;	// Used to test for a specific Stop Code to report to the Host
	bOverHeight					: BOOL; 	// Detect OverHeight to report to the Host
	st_UpdateMessageToSend		: ST_Item;			// Message to Send to Host

	fb_SorterUpdateBuffer			: FB_ItemBuffer;	// Function to Process the SorterUpdateBuffer

	fb_SorterTransportBuffer		: FB_ItemBuffer;	// Function to Process the SorterTransportBuffer

	sMessage	:	STRING;
	
END_VAR

VAR CONSTANT
	SEND_ARRIVAL			:	INT := 5;
	SEND_LOCATION			:	INT := 7;
	TransmitMsgBuffer_Size	:	INT :=	25;		// Number of Messages to hold in buffer
END_VAR

// Create instances of Buffer Processing Functions to initialize the buffers and data
fb_SorterUpdateBuffer.Master := TRUE;
fb_SorterTransportBuffer.Master := TRUE;

// Activate or de-activate logging
fb_SorterUpdateBuffer.LogEntries := .nItemBufferLogEnable.UPDATE;
fb_SorterTransportBuffer.LogEntries := .nItemBufferLogEnable.TRANSPORT;

// Setup Buffer names for Logging purposes
fb_SorterUpdateBuffer.Name := 'SYS UPDATE';
fb_SorterTransportBuffer.Name := 'SYS TRANSPORT';

fb_SorterUpdateBuffer(st_BufferData := st_SorterUpdateBuffer
					, st_BufferFdbkIn := st_UpdateFdbkIn
					, st_BufferFdbkOut => st_UpdateFdbkOut);
fb_SorterTransportBuffer(st_BufferData := st_SorterTransportBufferP6040
					, st_BufferFdbkIn := st_TransportFdbkInP6040
					, st_BufferFdbkOut => st_TransportFdbkOutP6040);

(* -------------------- On Receive Message Process the data -------------------- *)
IF RxCounter_Old <> ServerControl.fbServer.aApplications[nConnectionIndex].RxCounter  THEN
	ItemTransport := BlankItem; // Clear the ItemTransport each pass to capture only new transport commands
	RECEIVE();
	// Test the DeviceID and route the Transport accordingly
	//	If there is only one possible DeviceID, this IF statement can be removed, but the fb_(TransportBuffer).AddItem call still has to be made
	//	Also, the default destination needs to be passed per DeviceID
	IF DeviceID = Sorter.st_SorterCfg.EquipID THEN
		fb_SorterTransportBuffer.AddItem(st_ItemToAdd := ItemTransport);
		IF DefDestination <> 0 THEN 
 		GVL_SorterItems.P6040_DefaultDestination := DefDestination;
		END_IF
	END_IF
	RxCounter_Old := ServerControl.fbServer.aApplications[nConnectionIndex].RxCounter;
END_IF

(* -------------------- Transmit Messages if any are waiting in the buffer --------------------- *)
IF SendingMsg_Index <> TransmitMsgBuffer_Index THEN
	TRANSMIT(TransmitEnable:= TRUE);
END_IF

(* -------------------- Watch Bar code readers and send message when load is read -------------------- *)

(* ----- BCR10563: P6040_01 Divert 1 ----- *)	
ReadBCRID_S6040_01_Old := BarCodeMessage(cDatamanReader := BarCodeReaders.BCR_S6040_01
									, nOldCount := ReadBCRID_S6040_01_Old
									, nMessageToSend := SEND_ARRIVAL);
(* ----- BCR10564: P8015 Lane Confirm ----- *)	
ReadBCRID_S7004_01_Old := BarCodeMessage(cDatamanReader := BarCodeReaders.BCR_S7004_01
									, nOldCount := ReadBCRID_S7004_01_Old
									, nMessageToSend := SEND_LOCATION);


(* -------------------- Watch Sorter and Device Status and transmit on change -------------------- *)
// Transmit On update from Sorter
// Detect a new message to process when the in and out pointer values disagree
IF st_SorterUpdateBuffer.nInPointer <> fb_SorterUpdateBuffer.OutPointer THEN
	// Pull the next message out of the buffer
	fb_SorterUpdateBuffer.RemoveItem(st_ItemToReturn => st_UpdateMessageToSend);
	CASE st_UpdateMessageToSend.MessageType OF

		E_MessageIds.TransportResponse_25:			// Response to a Transport Command

			CASE st_UpdateMessageToSend.Status OF
				E_StatusCode.Assign_Accepted:		// Assignment Accepted
					TransmitMsgStatus := E_TransportResponse.Accepted; 
				E_StatusCode.Assign_Full:			// Assigned Lane Unavailable
					TransmitMsgStatus := E_TransportResponse.DivertLaneUnavailable; 
				E_StatusCode.Assign_NotFound:		// Assigned Load ID Not Found
					TransmitMsgStatus := E_TransportResponse.LoadIdNotFound; 
				E_StatusCode.Assign_NotInducted:	// Assigned Load Not Inducted
					TransmitMsgStatus := E_TransportResponse.NextLoadReady; 
				E_StatusCode.Diverting:	// Assigned Load already Inducting
					TransmitMsgStatus := E_TransportResponse.LateInduction; 
			ELSE
				TransmitMsgStatus := E_TransportResponse.UnknownFailure; // Capture any other failures
				IF nMessageLogEnable.TransportResponse_25 THEN
					sMessage := CONCAT(' Item: ', st_UpdateMessageToSend.ID);
					sMessage := CONCAT(sMessage,' Destination: ');
					sMessage := CONCAT(sMessage, DINT_TO_STRING(st_UpdateMessageToSend.Destination));
					sMessage := CONCAT(sMessage,' TR Status: ');
					sMessage := CONCAT(sMessage, DINT_TO_STRING(st_UpdateMessageToSend.Status));
					// Write to the Error List
					ADSLOGSTR( msgCtrlMask := ADSLOG_MSGTYPE_HINT OR ADSLOG_MSGTYPE_LOG
						, msgFmtStr := 'Unhandled Transport Response Status: %s'
						, strArg := sMessage);
				END_IF
			END_CASE
			TransmitMsgBuffer[TransmitMsgBuffer_Index] := TransportResponse(Device := st_UpdateMessageToSend.DeviceID
																			, Barcode := st_UpdateMessageToSend.ID
																			, Status := TransmitMsgStatus);
			TransmitMsgBuffer_Index := IncIndex(TransmitMsgBuffer_Index,1,TransmitMsgBuffer_Size);

		E_MessageIds.TransportComplete_26:			// Indication of the final disposition of a transported item

			CASE st_UpdateMessageToSend.Status OF
				E_StatusCode.Divert_Success:		// Divert Success Message
					TransmitMsgStatus := E_TransportComplete.Success; 
				E_StatusCode.Divert_Complete:		// Divert Success Message
					TransmitMsgStatus := E_TransportComplete.Success; 
			ELSE 									// Catch all other failures
				TransmitMsgStatus := E_TransportComplete.Faulted; 
			END_CASE			
			CASE st_UpdateMessageToSend.ExtStatus OF
				E_StatusCode.Divert_Full:			// Divert Full/Unavailable
					TransmitMsgStatus := E_TransportComplete.Unavailable; 
				E_StatusCode.Divert_Offline:		// Divert Offline
					TransmitMsgStatus := E_TransportComplete.Offline; 
				E_StatusCode.Divert_Missed:		// Divert Missed
					TransmitMsgStatus := E_TransportComplete.Passed; 
				E_StatusCode.Divert_Recirculated:		// Divert Missed
					TransmitMsgStatus := E_TransportComplete.Success; 
			END_CASE			
			TransmitMsgBuffer[TransmitMsgBuffer_Index] := TransportComplete(Device:= st_UpdateMessageToSend.DeviceID
																			, BarCode:= st_UpdateMessageToSend.ID
																			, Dest:= DINT_TO_INT(st_UpdateMessageToSend.Destination)
																			, Status:= TransmitMsgStatus ); 
			TransmitMsgBuffer_Index := IncIndex(TransmitMsgBuffer_Index,1,TransmitMsgBuffer_Size);

	END_CASE
END_IF

// Transmit on Device Status Change
DeviceStatus();

(* -------------------- Reset The Transmit Triger after the message is succesfully added to the buffer ------------------- *)
IF ((ServerControl.fbServer.aApplications[nConnectionIndex].bTransmitTrigger = TRUE) OR ServerControl.TransmitTrigger = TRUE)  AND (TxCounter_Old <> ServerControl.fbServer.aApplications[nConnectionIndex].TxCounter) THEN
	ServerControl.TransmitTrigger := FALSE;
	TRANSMIT(TransmitEnable:= FALSE);
	TxCounter_Old := ServerControl.fbServer.aApplications[nConnectionIndex].TxCounter;
END_IF

METHOD PRIVATE Arrival : STRING(55)
VAR_INPUT
	Device :	STRING(5);		// Device Label per communication standard
	BarCode:	STRING(30);		// Barcode from barcode reader
	DefDest:	INT;		// Default destination
END_VAR
VAR
	String1: STRING(55);
	BC_Len: INT;
	x: INT;
	String_DefDest: STRING(2);
	y: INT;
	Device_Len: INT;
	i: INT;
END_VAR
(* Message from communication Spec:
	[STX (0x02h)][23][Device ID (5 CHR)][Barcode (20 CHR)][Default Dest (2 CHR)][Blank (22 CHR)][ETX 0x03h)]
*)

// Start Message with header
String1 := '$0223';

// Check Device for length and Pad with spaces if needed
Device_Len := LEN(Device);
IF Device_Len = 5 THEN
	String1 := CONCAT(STRING1, Device);
ELSIF Device_Len < 5 THEN
	String1 := CONCAT(STRING1, Device);
	FOR i := 1 TO (5-Device_Len) DO
		String1 := CONCAT(String1,' ');
	END_FOR
ELSE
	String1 := CONCAT(String1, 'XXXXX');
END_IF

// Check Barcode for length and Pad with spaces if needed
BC_Len := LEN(BARCODE);
IF BC_Len <20 THEN
	String1 := CONCAT(STRING1, BarCode);
	FOR x := 1 TO (20-BC_Len) DO
		String1 := CONCAT(String1,' ');
	END_FOR
ELSIF BC_Len = 20 THEN
	String1 := CONCAT(STRING1, BarCode);
ELSE 
	String1 := CONCAT(STRING1, RIGHT(BarCode,20));	
END_IF

// Check Default Destination for length and Pad with spaces if needed
String_DefDest := INT_TO_STRING(DefDest);
IF DefDest < 10 THEN
	String1 := CONCAT(String1,'0');
	String1 := CONCAT(String1, String_DefDest);
ELSIF (DefDest >= 10) AND (DefDest < 100) THEN
	String1 := CONCAT(String1, String_DefDest);
ELSE
	String1 := CONCAT(String1, 'XX');
END_IF	

// Pad with spaces
FOR y := 1 TO 22 DO
	String1 := CONCAT(String1,' ');
END_FOR

// Add ending Character
String1 := CONCAT(String1,'$03');
	
Arrival := String1;
END_METHOD

METHOD PRIVATE BarCodeMessage : UDINT
VAR_INPUT
	cDatamanReader	: CognexDataMan260;
	//sLocation		:	STRING(5);
	nOldCount		:	UDINT;
	nMessageToSend	: 	INT;
END_VAR
IF nOldCount <> cDatamanReader.GoodreadCount THEN
	// Send location update message to host
	CASE nMessageToSend OF
		SEND_ARRIVAL:	TransmitMsgBuffer[TransmitMsgBuffer_Index] := Arrival(cDatamanReader.In_EquipID, cDatamanReader.Out_ReadString,00);
		SEND_LOCATION: TransmitMsgBuffer[TransmitMsgBuffer_Index] := LocationUpdate(cDatamanReader.In_EquipID, cDatamanReader.Out_ReadString,00);
	END_CASE
	TransmitMsgBuffer_Index := IncIndex(TransmitMsgBuffer_Index,1,TransmitMsgBuffer_Size);
	BarCodeMessage := cDatamanReader.GoodreadCount;
ELSE
	BarCodeMessage := nOldCount;
END_IF
END_METHOD

METHOD PRIVATE CustomMessage : UDINT
VAR_INPUT
	EquipID			: 	STRING(5);
	Barcode			:	STRING(30);
	nReadCount		:	UDINT;
	nOldCount		:	UDINT;
	nMessageToSend	: 	INT;
END_VAR
IF nOldCount <> nReadCount THEN
	// Send location update message to host
	CASE nMessageToSend OF
		SEND_ARRIVAL:	TransmitMsgBuffer[TransmitMsgBuffer_Index] := Arrival(EquipID, BarCode,00);
		SEND_LOCATION: TransmitMsgBuffer[TransmitMsgBuffer_Index] := LocationUpdate(EquipID, BarCode,00);
	END_CASE
	TransmitMsgBuffer_Index := IncIndex(TransmitMsgBuffer_Index,1,TransmitMsgBuffer_Size);
	CustomMessage := nReadCount;
ELSE
	CustomMessage := nOldCount;
END_IF
END_METHOD

ACTION DeviceStatus:
(*
	
	Local Data items used for Equipment status processing
	Msg_EquipStatArry:	ARRAY[1..7] OF ST_Msg_EquipStat;
	nSystemStatusIndex : INT; 	// Index used for Processing the system status array
	nEquipStatusIndex: INT;	//Index used for adding items to the MSG_EquipStatArray
	nTempOperState : DINT;	//Capture the Temporary Operating State of the Equipment for comparison
	
	GVL_EquipmentArray items used for Equipment Status processing
	// System Equipment
	SystemEquip_Count : INT; //Count of Equipment to Process in System PLC
	SystemEquipStatusArray : ARRAY[1..EQUIP_COUNT_MAX] OF ST_StateCntrlSts; //Array of Equipment Status Current
	SystemEquipStatusArray_Last : ARRAY[1..EQUIP_COUNT_MAX] OF ST_StateCntrlSts; //Array of Equipment Status Last State
*)

//===================================================================================
(* 	Process the Conveyor/Equipment status arrays comparing the current state to the last state
 	When a state change is deteted, add the correspoding equipment to the Msg_EquipStatArray
		Then increment/test the nEquipStatusIndex and add the message to the outbound buffer
		if the Msg_EquipStatArry is full, and reset the nEquipStatusIndex value to the lower bound
*)
// Initialise the nEquipStatusIndex to 0 to detect when items are in the Msg_EquipStatArry buffer
nEquipStatusIndex := 0;

FOR nSystemStatusIndex := 1 TO gvl_equiparrays.nSystemEquip_Count BY 1 DO
	// Test for a valid label, ignore if there isn't a label
	IF GVL_EquipArrays.aSystemEquipStatusArray[nSystemStatusIndex].Label <> '' THEN
		// Capture Offline State
		IF GVL_EquipArrays.aSystemEquipStatusArray[nSystemStatusIndex].CrntState = E_StateCntrl.stOffline THEN
			nTempOperState := E_OperStateCntrl.Offline;
		ELSE
			// Check for OverHeight
			// Initialise the stop register with the conveyor stop register
			fb_CheckStopRegister(aCodeRegister := GVL_EquipArrays.aSystemEquipStatusArray[nSystemStatusIndex].stsStopRegister);
			// Check for an OverHeight in the Stop Register
			fb_CheckStopRegister.Check(nCodeToCheck := E_StopCodes.OverHeightFLT,
				bCodeSet => bOverHeight);
			// Set over Height
			IF bOverHeight THEN
				nTempOperState := E_OperStateCntrl.OverHeight;
			ELSE
				// Capture Faulted State, or a specific Fault (in this instance, OverHeight)
				IF GVL_EquipArrays.aSystemEquipStatusArray[nSystemStatusIndex].CrntState = E_StateCntrl.stFaulted THEN
						nTempOperState := E_OperStateCntrl.Faulted;
				ELSE
					// Capture Auto/Manual States and Running/Sleeping states where appropriate
					IF GVL_EquipArrays.aSystemEquipStatusArray[nSystemStatusIndex].CrntState = E_StateCntrl.stAuto THEN
						// Capture Auto-Running
						IF GVL_EquipArrays.aSystemEquipStatusArray[nSystemStatusIndex].CrntOperState = E_OperStateCntrl.running THEN
							nTempOperState := E_OperStateCntrl.running;
						// Capture Auto-Sleeping
						ELSIF GVL_EquipArrays.aSystemEquipStatusArray[nSystemStatusIndex].CrntOperState = E_OperStateCntrl.sleeping THEN
							nTempOperState := E_OperStateCntrl.sleeping;
						// Capture Auto
						ELSE
							nTempOperState := E_OperStateCntrl.Auto;
						END_IF
					ELSE
						// Capture Manual-Running
						IF GVL_EquipArrays.aSystemEquipStatusArray[nSystemStatusIndex].CrntOperState = E_OperStateCntrl.running THEN
							nTempOperState := E_OperStateCntrl.running;
						// Capture Manual
						ELSE
							nTempOperState := E_OperStateCntrl.Manual;
						END_IF
					END_IF
				END_IF
			END_IF
		END_IF
		// Test for a change in Operational state or a non-initialized Storage array
		IF GVL_EquipArrays.aSystemEquipStatusArray_last[nSystemStatusIndex].LstOperState <> nTempOperState OR GVL_EquipArrays.aSystemEquipStatusArray_last[nSystemStatusIndex].Index = 0 THEN
			IF GVL_EquipArrays.aSystemEquipStatusArray_last[nSystemStatusIndex].Index = 0 THEN
				// Initialise the Storage Data Record
				GVL_EquipArrays.aSystemEquipStatusArray_last[nSystemStatusIndex] := GVL_EquipArrays.aSystemEquipStatusArray[nSystemStatusIndex];
			END_IF
			// Capture the nTempOperState for future comparisons
			GVL_EquipArrays.aSystemEquipStatusArray_last[nSystemStatusIndex].LstOperState := TO_INT(nTempOperState);
			// Increment the status index and check for roll-over
			nEquipStatusIndex := nEquipStatusIndex + 1;
			IF nEquipStatusIndex > 7 THEN
				// When there are 7 status updates, create the message
				TransmitMsgBuffer[TransmitMsgBuffer_Index] := EquipStatUpdate(Msg_EquipStatArry);
				// Increment the buffer index
				TransmitMsgBuffer_Index := IncIndex(TransmitMsgBuffer_Index,1,TransmitMsgBuffer_Size);
				// Set the index for the next message
				nEquipStatusIndex := 1;
			END_IF
			// Capture the Label and Index of the current Equipment status record
			Msg_EquipStatArry[nEquipStatusIndex].DeviceID := GVL_EquipArrays.aSystemEquipStatusArray[nSystemStatusIndex].Label;
			Msg_EquipStatArry[nEquipStatusIndex].Status := TO_INT(nTempOperState);
		END_IF
	END_IF
END_FOR

// Detect unsent items in the Msg_EquipStatArry buffer
IF nEquipStatusIndex > 0 THEN
	// Prepare the Equipment Status Message
	TransmitMsgBuffer[TransmitMsgBuffer_Index] := EquipStatUpdate(Msg_EquipStatArry);
	// Add the Equipment Status Message to the outbound buffer
	TransmitMsgBuffer_Index := IncIndex(TransmitMsgBuffer_Index,1,TransmitMsgBuffer_Size);
END_IF
END_ACTION

METHOD PRIVATE EquipStatUpdate : STRING(55)
VAR_IN_OUT
	Msg_ConveyorStatArry:	ARRAY[1..7] OF ST_Msg_EquipStat; // Array of Device status
END_VAR
VAR
	String1: STRING(55);
	x: INT;
	String_DefDest: STRING(2);
	y: INT;
	String_Status: STRING(2);
	Device_Len: INT;
	i: INT;
END_VAR
(* Message from communication Spec:
	[STX (0x02h)][28][Device 1 ID (5 CHR)][Status (2 CHR)] repeated for devices thru 7[ETX 0x03h)]
*)

// Start Message with header
String1 := '$0228';

FOR x := 1 TO 7 DO
	IF (Msg_ConveyorStatArry[x].DeviceID <> '') THEN
		// Check Device for length and Pad with spaces if needed
		Device_Len := LEN(Msg_ConveyorStatArry[x].DeviceID);
		IF Device_Len = 5 THEN
			String1 := CONCAT(String1,Msg_ConveyorStatArry[x].DeviceID);
		ELSIF Device_Len < 5 THEN
			Device_Len := LEN(Msg_ConveyorStatArry[x].DeviceID);
			FOR i := 1 TO (5-Device_Len) DO
				String1 := CONCAT(String1,' ');
			END_FOR
		ELSE
			String1 := CONCAT(String1, 'XXXXX');
		END_IF
		// Clear the DeviceID after processing
		Msg_ConveyorStatArry[x].DeviceID := '';
		
	
		// Check Status for length and Pad with spaces if needed
		String_Status := INT_TO_STRING(Msg_ConveyorStatArry[x].Status);
		IF Msg_ConveyorStatArry[x].Status < 10 THEN
			String1 := CONCAT(String1,'0');
			String1 := CONCAT(String1, String_Status);
		ELSIF (Msg_ConveyorStatArry[x].Status >= 10) AND (Msg_ConveyorStatArry[x].Status < 100) THEN
			String1 := CONCAT(String1, String_Status);
		ELSE
			String1 := CONCAT(String1, 'XX');
		END_IF	
		// Clear the Status after processing
		Msg_ConveyorStatArry[x].Status := 0;
	ELSE 
		String1 := CONCAT(String1,'       ');
	END_IF	
END_FOR

// Add ending Character
String1 := CONCAT(String1,'$03');
	
EquipStatUpdate := String1;
END_METHOD

METHOD PRIVATE KeepAliveResponse : STRING(55)
VAR_INPUT
END_VAR
VAR
	String1: STRING(55);
	x: INT;
END_VAR
(* Message from communication Spec:
	[STX (0x02h)][29][Blank (49 CHR)][ETX 0x03h)]
*)

// Start Message with header
String1 := '$0229';

// Pad with Spaces
FOR x := 1 TO 49 DO
	String1 := CONCAT(String1,' ');
END_FOR

// Add ending Character
String1 := CONCAT(String1,'$03');
	
KeepAliveResponse := String1;
END_METHOD

METHOD PRIVATE LocationUpdate : STRING(55)
VAR_INPUT
	Device :	STRING(5);		// Device Label per communication standard
	BarCode:	STRING(30);		// Barcode from barcode reader
	Dest:	INT;		// Default destination
END_VAR
VAR
	String1: STRING(55);
	BC_Len: INT;
	x: INT;
	String_Dest: STRING(2);
	y: INT;
	Device_Len: INT;
	i: INT;
END_VAR
(* Message from communication Spec:
	[STX (0x02h)][27][Device ID (5 CHR)][Barcode (20 CHR)][Destination (2 CHR)][Blank (24 CHR)][ETX 0x03h)]
*)

// Start Message with header
String1 := '$0227';

// Check Device for length and Pad with spaces if needed
Device_Len := LEN(Device);
IF Device_Len = 5 THEN
	String1 := CONCAT(STRING1, Device);
ELSIF Device_Len < 5 THEN
	String1 := CONCAT(STRING1, Device);
	FOR i := 1 TO (5-Device_Len) DO
		String1 := CONCAT(String1,' ');
	END_FOR	
ELSE
	String1 := CONCAT(String1, 'XXXXX');
END_IF


// Check Barcode for length and Pad with spaces if needed
BC_Len := LEN(BARCODE);
IF BC_Len <20 THEN
	String1 := CONCAT(STRING1, BarCode);
	FOR x := 1 TO (20-BC_Len) DO
		String1 := CONCAT(String1,' ');
	END_FOR
ELSIF BC_Len = 20 THEN
	String1 := CONCAT(STRING1, BarCode);
ELSE 
	String1 := CONCAT(STRING1, RIGHT(BarCode,20));	
END_IF

(* Destination isn't needed in location Update 
// Check Default Destination for length and Pad with spaces if needed
String_Dest := INT_TO_STRING(Dest);
IF Dest < 10 THEN
	String1 := CONCAT(String1,'0');
	String1 := CONCAT(String1, String_Dest);
ELSIF (Dest >= 10) AND (Dest < 100) THEN
	String1 := CONCAT(String1, String_Dest);
ELSE
	String1 := CONCAT(String1, 'XX');
END_IF	
*)

// Pad with spaces
FOR y := 1 TO 24 DO
	String1 := CONCAT(String1,' ');
END_FOR

// Add ending Character
String1 := CONCAT(String1,'$03');
	
LocationUpdate := String1;
END_METHOD

ACTION RECEIVE:
// Empty all outputs
	DeviceID := BarCode := '';
	Destination := DefDestination := 0;
	Status := 99;
	Msg_EquipStatArry := Blank_Msg_ConveyorStatArry;

	// Set up index with clipping to keep it within array boundaries	
	i := IncIndex(i,1,10);
		
	// Clear one before to make it easy to find newest entry 
	IF i = 10 THEN
		RawMsgArray[1] := '';	
		RawMsgLenArray[1] := 0;	
		RawMsgStartPosArray[1] := 0;
		RawMsgEndPosArray[1] :=  0;
	ELSE
		RawMsgArray[i+1] := '';	
		RawMsgLenArray[i+1] := 0;	
		RawMsgStartPosArray[i+1] := 0;
		RawMsgEndPosArray[i+1] :=  0;
	END_IF
	
	
	// Fill Appropriate info for each message
	RawMsgArray[i] := ServerControl.fbServer.aApplications[nConnectionIndex].RxRawMessage;	
	RawMsgLenArray[i] := LEN(ServerControl.fbServer.aApplications[nConnectionIndex].RxRawMessage);	
	StrStartPos := FIND(STR1:= RawMsgArray[i], STR2:='$02' );
	StrEndPos :=  FIND(STR1:= RawMsgArray[i], STR2:='$03' );
	RawMsgStartPosArray[i] := StrStartPos;
	RawMsgEndPosArray[i] := StrEndPos;
	
{info 'Maybe: Possibly add do while loop here to process the case where more than one message comes in at a time and clean up StrStartPos and end pos with array'}	
	IF StrStartPos <> 0 THEN
		MsgString := MID(STR:=ServerControl.fbServer.aApplications[nConnectionIndex].RxRawMessage , LEN:= 51 , POS:= StrStartPos);
		MsgArray[i] := MsgString;
		MsgID := STRING_TO_DINT(MID(STR:=ServerControl.fbServer.aApplications[nConnectionIndex].RxRawMessage , LEN:= 2, POS:= StrStartPos+1));
	
		CASE MsgID OF
			E_MessageIds.TransportCommand_05:  	// Transport Command Message
				DeviceID := MID(STR:=ServerControl.fbServer.aApplications[nConnectionIndex].RxRawMessage, LEN:= 5, POS:= StrStartPos+3);
				BarCode := MID(STR:=ServerControl.fbServer.aApplications[nConnectionIndex].RxRawMessage, LEN:= 20, POS:= StrStartPos+8);
				Destination := STRING_TO_DINT( MID(STR:=ServerControl.fbServer.aApplications[nConnectionIndex].RxRawMessage, LEN:= 2, POS:= StrStartPos+28));
				DefDestination := STRING_TO_DINT( MID(STR:=ServerControl.fbServer.aApplications[nConnectionIndex].RxRawMessage, LEN:= 2, POS:= StrStartPos+30));
				Status := STRING_TO_BYTE( MID(STR:=ServerControl.fbServer.aApplications[nConnectionIndex].RxRawMessage , LEN:= 2, POS:= StrStartPos+50));

				//Strip spaces from Bar Code
				SpacePosition := (FIND(STR1:= BarCode, STR2:=' ' ))+3;
				BarCodeNoSpace := MID(STR:=BarCode, LEN:= (20-SpacePosition), POS:= 1);
				// Update Info to send to Sorter PLC
//				ItemTransport := BlankItem;
				ItemTransport.DeviceID := DeviceID;
				ItemTransport.ID := BarCodeNoSpace;
				ItemTransport.Destination := Destination;
				ItemTransport.Status := E_StatusCode.UpdateNeeded;
				ItemTransport.MessageType := E_MessageIds.TransportCommand_05;
//				fb_SorterTransportBuffer.AddItem(st_ItemToAdd := ItemTransport);
//				Out_DefaultDestination := DefDestination;

			E_MessageIds.LocationUpdateResponse_07:		// Location Update Response
				DeviceID := MID(STR:=ServerControl.fbServer.aApplications[nConnectionIndex].RxRawMessage , LEN:= 5, POS:= StrStartPos+3);
				BarCode := MID(STR:=ServerControl.fbServer.aApplications[nConnectionIndex].RxRawMessage , LEN:= 20, POS:= StrStartPos+8);
				Destination := STRING_TO_DINT( MID(STR:=ServerControl.fbServer.aApplications[nConnectionIndex].RxRawMessage , LEN:= 2, POS:= StrStartPos+23));
				Status := STRING_TO_BYTE( MID(STR:=ServerControl.fbServer.aApplications[nConnectionIndex].RxRawMessage , LEN:= 2, POS:= StrStartPos+50));
						
			E_MessageIds.EquipmentStatusResponse_08:		// Equipment Status Response
				FOR j := 0 TO 6 DO
					Msg_EquipStatArry[j+1].DeviceID := MID(STR:=ServerControl.fbServer.aApplications[nConnectionIndex].RxRawMessage , LEN:= 5, POS:= ((StrStartPos+3)+(j*7)));
					Msg_EquipStatArry[j+1].Status := STRING_TO_BYTE(MID(STR:=ServerControl.fbServer.aApplications[nConnectionIndex].RxRawMessage , LEN:= 2, POS:= ((StrStartPos+8)+(j*7))));	
				END_FOR
			
			E_MessageIds.KeepAlive_09:		// Keep Alive
				// If Keep Alive message is recieved send the response to the transmit buffer
				TransmitMsgBuffer[TransmitMsgBuffer_Index] := KeepAliveResponse();
				TransmitMsgBuffer_Index := IncIndex(TransmitMsgBuffer_Index,1,TransmitMsgBuffer_Size);				
		END_CASE
	END_IF
END_ACTION

ACTION TRANSMIT:

// Transmit messages from buffer
IF NOT ServerControl.TransmitTrigger AND TransmitEnable THEN
	ServerControl.TxMessage := TransmitMsgBuffer[SendingMsg_Index];
	ServerControl.TransmitTrigger := TRUE;
	SendingMsg_Index := IncIndex(SendingMsg_Index,1,TransmitMsgBuffer_Size);
	
	TransmittedArray[y] := ServerControl.TxMessage;
	// Clear out message before last update to ease in testing
	IF y = 10 THEN
		TransmittedArray[1] := '';
	ELSE
		TransmittedArray[y+1] := '';
	END_IF
	
	y :=  IncIndex(IDX:= y, IdxMIN:= 0, IdxMAX:=10 );
END_IF
END_ACTION

METHOD PRIVATE TransportComplete : STRING(55)
VAR_INPUT
	Device :	STRING(5);		// Device Label per communication standard
	BarCode:	STRING(30);		// Barcode from barcode reader
	Dest:	INT;		// Default destination
	Status:	INT;		// Status
END_VAR
VAR
	String1: STRING(55);
	BC_Len: INT;
	x: INT;
	String_Dest: STRING(2);
	y: INT;
	String_Status: STRING(2);
	Device_Len: INT;
	i: INT;
END_VAR
(* Message from communication Spec:
	[STX (0x02h)][26][Device ID (5 CHR)][Barcode (20 CHR)][Destination (2 CHR)][Blank (20 CHR)][Status (2 CHR)][ETX 0x03h)]
*)

// Start Message with header
String1 := '$0226';

// Check Device for length and Pad with spaces if needed
Device_Len := LEN(Device);
IF Device_Len = 5 THEN
	String1 := CONCAT(STRING1, Device);
ELSIF Device_Len < 5 THEN
	String1 := CONCAT(STRING1, Device);
	FOR i := 1 TO (5-Device_Len) DO
		String1 := CONCAT(String1,' ');
	END_FOR
ELSE
	String1 := CONCAT(String1, 'XXXXX');
END_IF

// Check Barcode for length and Pad with spaces if needed
BC_Len := LEN(BARCODE);
IF BC_Len <20 THEN
	String1 := CONCAT(STRING1, BarCode);
	FOR x := 1 TO (20-BC_Len) DO
		String1 := CONCAT(String1,' ');
	END_FOR
ELSIF BC_Len = 20 THEN
	String1 := CONCAT(STRING1, BarCode);
ELSE 
	String1 := CONCAT(STRING1, RIGHT(BarCode,20));	
END_IF

// Check Destination for length and Pad with spaces if needed
String_Dest := INT_TO_STRING(Dest);
IF Dest < 10 THEN
	String1 := CONCAT(String1,'0');
	String1 := CONCAT(String1, String_Dest);
ELSIF (Dest >= 10) AND (Dest < 100) THEN
	String1 := CONCAT(String1, String_Dest);
ELSE
	String1 := CONCAT(String1, 'XX');
END_IF	

// Pad with Spaces
FOR y := 1 TO 20 DO
	String1 := CONCAT(String1,' ');
END_FOR

// Check Status for length and Pad with spaces if needed
String_Status := INT_TO_STRING(Status);
IF Status < 10 THEN
	String1 := CONCAT(String1,'0');
	String1 := CONCAT(String1, String_Status);
ELSIF (Status >= 10) AND (Status < 100) THEN
	String1 := CONCAT(String1, String_Status);
ELSE
	String1 := CONCAT(String1, 'XX');
END_IF	

// Add ending Character
String1 := CONCAT(String1,'$03');
	
TransportComplete := String1;
END_METHOD

METHOD PRIVATE TransportResponse : STRING(55)
VAR_INPUT
	Device :	STRING(5);		// Device Label per communication standard
	BarCode :	STRING(30);		// Barcode from barcode reader
	Status :	INT;		// Status
END_VAR
VAR
	String1: STRING(55);
	BC_Len: INT;
	x: INT;
	String_Status: STRING(2);
	y: INT;
	Device_Len: INT;
	i: INT;
END_VAR
(* Message from communication Spec:
	[STX (0x02h)][25][Device ID (5 CHR)][Barcode (20 CHR)][Blank (22 CHR)][Status (2 CHR)][ETX 0x03h)]
*)

// Start Message with header
String1 := '$0225';

// Check Device for length and Pad with spaces if needed
Device_Len := LEN(Device);
IF Device_Len = 5 THEN
	String1 := CONCAT(STRING1, Device);
ELSIF Device_Len < 5 THEN
	String1 := CONCAT(STRING1, Device);
	FOR i := 1 TO (5-Device_Len) DO
		String1 := CONCAT(String1,' ');
	END_FOR
ELSE
	String1 := CONCAT(String1, 'XXXXX');
END_IF

// Check Barcode for length and Pad with spaces if needed
BC_Len := LEN(BARCODE);
IF BC_Len <20 THEN
	String1 := CONCAT(STRING1, BarCode);
	FOR x := 1 TO (20-BC_Len) DO
		String1 := CONCAT(String1,' ');
	END_FOR
ELSIF BC_Len = 20 THEN
	String1 := CONCAT(STRING1, BarCode);
ELSE 
	String1 := CONCAT(STRING1, RIGHT(BarCode,20));	
END_IF

// Pad with Spaces
FOR y := 1 TO 22 DO
	String1 := CONCAT(String1,' ');
END_FOR

// Check Status for length and Pad with spaces if needed
String_Status := INT_TO_STRING(Status);
IF Status < 10 THEN
	String1 := CONCAT(String1,'0');
	String1 := CONCAT(String1, String_Status);
ELSIF (Status >= 10) AND (Status < 100) THEN
	String1 := CONCAT(String1, String_Status);
ELSE
	String1 := CONCAT(String1, 'XX');
END_IF

// Add ending Character
String1 := CONCAT(String1,'$03');
	
TransportResponse := String1;
END_METHOD

END_PROGRAM

// ---- POUs/Log_Diverts.TcPOU
PROGRAM Log_Diverts
VAR
	r_DivertExtend			: ARRAY [1..16] OF R_TRIG;
	f_DivertExtend			: ARRAY [1..16] OF F_TRIG;
	r_ConfirmPE				: ARRAY [1..16] OF R_TRIG;
	f_ConfirmPE				: ARRAY [1..16] OF F_TRIG;
	sMessage				: STRING;
END_VAR

// Divert 1
r_DivertExtend[1](CLK := SORTER.aSorterDiverts[1].Output1);
f_DivertExtend[1](CLK := SORTER.aSorterDiverts[1].Output1);

IF r_DivertExtend[1].Q THEN
	IF .nDivertLogEnable.DIVERT1 THEN
		ADSLOGSTR( msgCtrlMask := ADSLOG_MSGTYPE_HINT OR ADSLOG_MSGTYPE_LOG
			, msgFmtStr := 'Extend Divert 1 : %s'
			, strArg := UDINT_TO_STRING(SORTER.st_SorterEncoder.CurrentCount)); 
	END_IF;
END_IF
IF f_DivertExtend[1].Q THEN
	IF .nDivertLogEnable.DIVERT1 THEN
		ADSLOGSTR( msgCtrlMask := ADSLOG_MSGTYPE_HINT OR ADSLOG_MSGTYPE_LOG
			, msgFmtStr := 'Retract Divert 1 : %s'
			, strArg := UDINT_TO_STRING(SORTER.st_SorterEncoder.CurrentCount)); 
	END_IF;
END_IF

// Confirm 1
r_ConfirmPE[1](CLK := SORTER.aSorterDiverts[1].ConfirmPE);
f_ConfirmPE[1](CLK := SORTER.aSorterDiverts[1].ConfirmPE);

IF r_ConfirmPE[1].Q THEN
	IF .nDivertLogEnable.CONFIRM1 THEN
		ADSLOGSTR( msgCtrlMask := ADSLOG_MSGTYPE_HINT OR ADSLOG_MSGTYPE_LOG
			, msgFmtStr := 'Confirm PE 1 Blocked: %s'
			, strArg := UDINT_TO_STRING(SORTER.st_SorterEncoder.CurrentCount)); 
	END_IF;
END_IF
IF f_ConfirmPE[1].Q THEN
	IF .nDivertLogEnable.CONFIRM1 THEN
		ADSLOGSTR( msgCtrlMask := ADSLOG_MSGTYPE_HINT OR ADSLOG_MSGTYPE_LOG
			, msgFmtStr := 'Confirm PE 1 Clear: %s'
			, strArg := UDINT_TO_STRING(SORTER.st_SorterEncoder.CurrentCount)); 
	END_IF;
END_IF

// Divert 2
r_DivertExtend[2](CLK := SORTER.aSorterDiverts[2].Output1);
f_DivertExtend[2](CLK := SORTER.aSorterDiverts[2].Output1);

IF r_DivertExtend[2].Q THEN
	IF .nDivertLogEnable.DIVERT2 THEN
		ADSLOGSTR( msgCtrlMask := ADSLOG_MSGTYPE_HINT OR ADSLOG_MSGTYPE_LOG
			, msgFmtStr := 'Extend Divert 2: %s'
			, strArg := UDINT_TO_STRING(SORTER.st_SorterEncoder.CurrentCount)); 
	END_IF;
END_IF
IF f_DivertExtend[2].Q THEN
	IF .nDivertLogEnable.DIVERT2 THEN
		ADSLOGSTR( msgCtrlMask := ADSLOG_MSGTYPE_HINT OR ADSLOG_MSGTYPE_LOG
			, msgFmtStr := 'Retract Divert 2: %s'
			, strArg := UDINT_TO_STRING(SORTER.st_SorterEncoder.CurrentCount)); 
	END_IF;
END_IF

// Confirm 2
r_ConfirmPE[2](CLK := SORTER.aSorterDiverts[2].ConfirmPE);
f_ConfirmPE[2](CLK := SORTER.aSorterDiverts[2].ConfirmPE);

IF r_ConfirmPE[2].Q THEN
	IF .nDivertLogEnable.CONFIRM2 THEN
		ADSLOGSTR( msgCtrlMask := ADSLOG_MSGTYPE_HINT OR ADSLOG_MSGTYPE_LOG
			, msgFmtStr := 'Confirm PE 2 Blocked: %s'
			, strArg := UDINT_TO_STRING(SORTER.st_SorterEncoder.CurrentCount)); 
	END_IF;
END_IF
IF f_ConfirmPE[2].Q THEN
	IF .nDivertLogEnable.CONFIRM2 THEN
		ADSLOGSTR( msgCtrlMask := ADSLOG_MSGTYPE_HINT OR ADSLOG_MSGTYPE_LOG
			, msgFmtStr := 'Confirm PE 2 Clear: %s'
			, strArg := UDINT_TO_STRING(SORTER.st_SorterEncoder.CurrentCount)); 
	END_IF
END_IF

// Sorter Discharge "Divert"
// Divert 3
r_DivertExtend[3](CLK := SORTER.aSorterDiverts[3].Output1);
f_DivertExtend[3](CLK := SORTER.aSorterDiverts[3].Output1);

IF r_DivertExtend[3].Q THEN
	IF .nDivertLogEnable.DIVERT3 THEN
		ADSLOGSTR( msgCtrlMask := ADSLOG_MSGTYPE_HINT OR ADSLOG_MSGTYPE_LOG
			, msgFmtStr := 'Extend Divert 3: %s'
			, strArg := UDINT_TO_STRING(SORTER.st_SorterEncoder.CurrentCount)); 
	END_IF;
END_IF
IF f_DivertExtend[3].Q THEN
	IF .nDivertLogEnable.DIVERT3 THEN
		ADSLOGSTR( msgCtrlMask := ADSLOG_MSGTYPE_HINT OR ADSLOG_MSGTYPE_LOG
			, msgFmtStr := 'Retract Divert 3: %s'
			, strArg := UDINT_TO_STRING(SORTER.st_SorterEncoder.CurrentCount)); 
	END_IF;
END_IF

// Confirm 3
r_ConfirmPE[3](CLK := SORTER.aSorterDiverts[3].ConfirmPE);
f_ConfirmPE[3](CLK := SORTER.aSorterDiverts[3].ConfirmPE);

IF r_ConfirmPE[3].Q THEN
	IF .nDivertLogEnable.CONFIRM3 THEN
		ADSLOGSTR( msgCtrlMask := ADSLOG_MSGTYPE_HINT OR ADSLOG_MSGTYPE_LOG
			, msgFmtStr := 'Confirm PE 3 Blocked: %s'
			, strArg := UDINT_TO_STRING(SORTER.st_SorterEncoder.CurrentCount)); 
	END_IF;
END_IF
IF f_ConfirmPE[3].Q THEN
	IF .nDivertLogEnable.CONFIRM3 THEN
		ADSLOGSTR( msgCtrlMask := ADSLOG_MSGTYPE_HINT OR ADSLOG_MSGTYPE_LOG
			, msgFmtStr := 'Confirm PE 3 Clear: %s'
			, strArg := UDINT_TO_STRING(SORTER.st_SorterEncoder.CurrentCount)); 
	END_IF
END_IF

// Divert 4
r_DivertExtend[4](CLK := SORTER.aSorterDiverts[4].Output1);
f_DivertExtend[4](CLK := SORTER.aSorterDiverts[4].Output1);

IF r_DivertExtend[4].Q THEN
	IF .nDivertLogEnable.DIVERT1 THEN
		ADSLOGSTR( msgCtrlMask := ADSLOG_MSGTYPE_HINT OR ADSLOG_MSGTYPE_LOG
			, msgFmtStr := 'Extend Divert 4 : %s'
			, strArg := UDINT_TO_STRING(SORTER.st_SorterEncoder.CurrentCount)); 
	END_IF;
END_IF
IF f_DivertExtend[4].Q THEN
	IF .nDivertLogEnable.DIVERT1 THEN
		ADSLOGSTR( msgCtrlMask := ADSLOG_MSGTYPE_HINT OR ADSLOG_MSGTYPE_LOG
			, msgFmtStr := 'Retract Divert 4 : %s'
			, strArg := UDINT_TO_STRING(SORTER.st_SorterEncoder.CurrentCount)); 
	END_IF;
END_IF

// Confirm 1
r_ConfirmPE[4](CLK := SORTER.aSorterDiverts[4].ConfirmPE);
f_ConfirmPE[4](CLK := SORTER.aSorterDiverts[4].ConfirmPE);

IF r_ConfirmPE[4].Q THEN
	IF .nDivertLogEnable.CONFIRM1 THEN
		ADSLOGSTR( msgCtrlMask := ADSLOG_MSGTYPE_HINT OR ADSLOG_MSGTYPE_LOG
			, msgFmtStr := 'Confirm PE 4 Blocked: %s'
			, strArg := UDINT_TO_STRING(SORTER.st_SorterEncoder.CurrentCount)); 
	END_IF;
END_IF
IF f_ConfirmPE[4].Q THEN
	IF .nDivertLogEnable.CONFIRM1 THEN
		ADSLOGSTR( msgCtrlMask := ADSLOG_MSGTYPE_HINT OR ADSLOG_MSGTYPE_LOG
			, msgFmtStr := 'Confirm PE 4 Clear: %s'
			, strArg := UDINT_TO_STRING(SORTER.st_SorterEncoder.CurrentCount)); 
	END_IF;
END_IF

// Divert 5
r_DivertExtend[5](CLK := SORTER.aSorterDiverts[5].Output1);
f_DivertExtend[5](CLK := SORTER.aSorterDiverts[5].Output1);

IF r_DivertExtend[5].Q THEN
	IF .nDivertLogEnable.DIVERT1 THEN
		ADSLOGSTR( msgCtrlMask := ADSLOG_MSGTYPE_HINT OR ADSLOG_MSGTYPE_LOG
			, msgFmtStr := 'Extend Divert 5 : %s'
			, strArg := UDINT_TO_STRING(SORTER.st_SorterEncoder.CurrentCount)); 
	END_IF;
END_IF
IF f_DivertExtend[5].Q THEN
	IF .nDivertLogEnable.DIVERT1 THEN
		ADSLOGSTR( msgCtrlMask := ADSLOG_MSGTYPE_HINT OR ADSLOG_MSGTYPE_LOG
			, msgFmtStr := 'Retract Divert 5 : %s'
			, strArg := UDINT_TO_STRING(SORTER.st_SorterEncoder.CurrentCount)); 
	END_IF;
END_IF

// Confirm 5
r_ConfirmPE[5](CLK := SORTER.aSorterDiverts[5].ConfirmPE);
f_ConfirmPE[5](CLK := SORTER.aSorterDiverts[5].ConfirmPE);

IF r_ConfirmPE[5].Q THEN
	IF .nDivertLogEnable.CONFIRM1 THEN
		ADSLOGSTR( msgCtrlMask := ADSLOG_MSGTYPE_HINT OR ADSLOG_MSGTYPE_LOG
			, msgFmtStr := 'Confirm PE 5 Blocked: %s'
			, strArg := UDINT_TO_STRING(SORTER.st_SorterEncoder.CurrentCount)); 
	END_IF;
END_IF
IF f_ConfirmPE[5].Q THEN
	IF .nDivertLogEnable.CONFIRM1 THEN
		ADSLOGSTR( msgCtrlMask := ADSLOG_MSGTYPE_HINT OR ADSLOG_MSGTYPE_LOG
			, msgFmtStr := 'Confirm PE 5 Clear: %s'
			, strArg := UDINT_TO_STRING(SORTER.st_SorterEncoder.CurrentCount)); 
	END_IF;
END_IF

END_PROGRAM

// ---- POUs/P_PulseCountDist.TcPOU
PROGRAM P_PulseCountDist
VAR
	EncoderValue : UDINT;
	StartValue: UDINT;
	EndValue: UDINT;
	Reading: BOOL;
	TotalCounts: UDINT;
	ReadCount: UDINT;
	ReadSum: UDINT;
	ReadAvg: REAL;
	Reset: BOOL;
	Timer: TON;
	TimeElapsed: REAL;
	Distance : REAL;
	Speed_ips : REAL;
	Speed_fps : REAL;
	Speed_fpm : REAL;
	DistperCount :	REAL;
	TestStart: R_TRIG;
	TestEnd: R_TRIG;
END_VAR

VAR CONSTANT
	EncoderMax: UDINT := Sorter.SORTERENCODERMAX;
END_VAR

// Uncomment to get pulse counts for a distance
TestStart(CLK:= (* Start photo eye goes here --> *) Photoeyes.PE_7171.Out);
TestEnd(CLK:= (* End photo eye goes here --> *) Photoeyes.PE_8211.Out);
EncoderValue := GVL_IO.ENC_9021_Raw;

Timer(IN:= Reading, PT:= T#1H, Q=> , ET=> );

IF Reset THEN
	ReadCount := 0;	
	ReadSum := 0;
	ReadAvg := 0;
	Reset := FALSE;
END_IF

IF TestStart.Q THEN 
	StartValue := EncoderValue;
	Reading := TRUE;
	ReadCount := ReadCount +1;
END_IF

IF Reading THEN
	TimeElapsed := (TIME_TO_REAL(Timer.ET))/1000;
END_IF

IF TestEnd.Q THEN 
	EndValue := EncoderValue;
	IF EndValue < StartValue THEN
		TotalCounts := EncoderMax - StartValue;
		TotalCounts := TotalCounts + EndValue;
	ELSE
  		TotalCounts := (EndValue-StartValue);
	END_IF
	
	ReadSum := ReadSum + TotalCounts;
	IF  ReadCount > 0 THEN 
		ReadAvg := UDINT_TO_REAL(ReadSum)/UDINT_TO_REAL(ReadCount);
	END_IF
	 
	IF TimeElapsed > 0 THEN
		Speed_ips := (Distance/TimeElapsed);
		Speed_fps := Speed_ips/12;
		Speed_fpm := Speed_fps*60;
	END_IF
	IF TotalCounts > 0 THEN
		DistperCount := Distance / UDINT_TO_REAL(TotalCounts);
	END_IF
		Reading := FALSE;
END_IF

END_PROGRAM

// ---- POUs/ProcessBuffers_6040.TcPOU
PROGRAM ProcessBuffers_6040
VAR_IN_OUT
	st_NextToInduct					: ST_ItemTemporary;
	st_UpdateItem					: ST_ItemTemporary;
	st_TempInductItem				: ST_ItemTemporary;
	{attribute 'OPC.UA.DA' := '0'}
	st_Sorter						: ST_Sorter;
	{attribute 'OPC.UA.DA' := '0'}
	aDiverts						: ARRAY[Sorter.DIVERTMIN..Sorter.NUMBEROFDIVERTS] OF ST_DIVERT;
	aItems 							: ARRAY[Sorter.SORTERENCODERMIN..Sorter.SORTERENCODERMAX] OF ST_Item;
END_VAR

VAR_INPUT
	DestinationOverride				: DINT;	// Pass in Divert to sent item to regardless of the direction received
	DivertToCommission				: DINT;
	ItemsArrayMax 					: UDINT;
	ItemsArrayMin 					: UDINT;
END_VAR

VAR_OUTPUT
	DefaultDestIdx					: DINT;
	RecircDestIdx					: DINT;
END_VAR

VAR
	fb_ArrivalBuffer				: FB_ItemBuffer;
	st_ArrivalItem 					: ST_Item;		// Arrival Item (Bar code read) from System PLC (BarCodeReaders.pou)

	// Item to replace in the sorter buffer
	st_ReplaceItem					: st_Item;

	fb_TransportBuffer				: FB_ItemBuffer;

	fb_UpdateBuffer 				: FB_ItemBuffer;

	st_ToUpdate						: ST_ItemTemporary;	// Item to Update on the Sorter, or waiting to be added to the sorter

	ItemsArraySize			: UDINT;

	TransportItemInSorter	: ST_Item;	// Temporary Processing Item
	TransportItemFound		: ST_Item;	// Item to Update Found
	TransportSorterIndex	: UDINT;

	ExitSorterIndex			: UDINT;
	ExitItemInSorter		: ST_Item;
	ExitItemFound			: ST_ItemTemporary;
	ExitInDivert			: BOOL;
	ExitDiverting			: BOOL;
	ExitSuccess				: BOOL;
	ExitDetected			: BOOL;
	ExitComplete			: BOOL;

	UpdateIndexCounter		: DINT;

	bTest : BOOL;
	sMessage	:	STRING;
	
	st_DisplayItem		:st_Item;
	LogSorterDump		:BOOL := FALSE;
	
	fb_FindDestination		: FB_FindDestination;
	fb_DefaultDestination	: FB_FindDestination;
	fb_RecircDestination	: FB_FindDestination;
	// Created to allow the aDiverts to be used in the FB_FindDestination Function Block
	{attribute 'OPC.UA.DA' := '0'}
	aTempDiverts			: ARRAY[Sorter.DIVERTMIN..Sorter.NUMBEROFDIVERTS] OF ST_DIVERT;

	nItemBufferLogEnable	:	UDINT;
	nSorterLogEnable		:	UDINT;
	nDivertLogEnable		:	UDINT;
	nSortBufferLogEnable	:	UDINT;
END_VAR

nItemBufferLogEnable := GVL_Logging.nItemBufferLogEnable OR GVL_Logging.nItemBufferLogEnable;
nSorterLogEnable := GVL_Logging.nSorterLogEnable OR GVL_Logging.nSorterLogEnable;
nDivertLogEnable := GVL_Logging.nDivertLogEnable OR GVL_Logging.nDivertLogEnable;
nSortBufferLogEnable := GVL_Logging.nSortBufferLogEnable OR GVL_Logging.nSortBufferLogEnable;

aTempDiverts := aDiverts;
// Initialize the Transport and Update buffers
// Set Master for FB's that control the buffer
fb_ArrivalBuffer.Master := FALSE;
fb_TransportBuffer.Master := FALSE;
fb_UpdateBuffer.Master := FALSE;

// Turn ON/OFF Logging of all activity in/out
fb_ArrivalBuffer.LogEntries := nItemBufferLogEnable.ARRIVALS;
fb_TransportBuffer.LogEntries := nItemBufferLogEnable.TRANSPORT;
fb_UpdateBuffer.LogEntries := nItemBufferLogEnable.UPDATE;

// Provide names for the buffers
fb_ArrivalBuffer.Name := CONCAT(st_Sorter.Config.Name, ' SRT ARRIVAL');
fb_TransportBuffer.Name := CONCAT(st_Sorter.Config.Name, ' SRT TRANSPORT');
fb_UpdateBuffer.Name := CONCAT(st_Sorter.Config.Name, ' SRT UPDATE');

// Initialize the FB_ItemExtBuffer Instances
fb_ArrivalBuffer(st_BufferData := st_SorterArrivalBufferP6040
						, st_BufferFdbkIn := st_ArrivalFdbkOutP6040
						, st_BufferFdbkOut => st_ArrivalFdbkInP6040);
fb_TransportBuffer(st_BufferData := st_SorterTransportBufferP6040
						, st_BufferFdbkIn := st_TransportFdbkOutP6040
						, st_BufferFdbkOut => st_TransportFdbkInP6040);
fb_UpdateBuffer(st_BufferData := st_SorterUpdateBuffer
						, st_BufferFdbkIn := st_UpdateFdbkOut
						, st_BufferFdbkOut => st_UpdateFdbkIn);

IF GVL_IO.INIT THEN
	fb_ArrivalBuffer.Clear();
	fb_TransportBuffer.Clear();
	fb_UpdateBuffer.Clear();
END_IF
						
(*
	Set the Upper/Lower bound of relevant arrays for looping purposes
	ItemsArrayMax/Min for the sorter array slot count
*)
// Size is Max - Min + 1 to capture both extremes
ItemsArraySize := ItemsArrayMax - ItemsArrayMin + 1;

(*
 	Check for a value disagreement in the Arrival Buffer In and Out pointers to
  	determine if there is an update for an item.
	When an Item arrives, the System PLC adds it to the shared buffer and increments
	the InPointer
*)
IF st_SorterArrivalBufferP6040.nInPointer <> fb_ArrivalBuffer.OutPointer THEN
	fb_ArrivalBuffer.RemoveItem(st_ItemToReturn => st_ArrivalItem);
END_IF

// Input Item read at bar code reader from System PLC to sorter
IF st_ArrivalItem.ID <> '' THEN
	IF nSortBufferLogEnable.BUFFER_ARRIVAL THEN
		sMessage := CONCAT('Item: ', st_ArrivalItem.ID);
		sMessage := CONCAT(sMessage,' Pulses: ');
		sMessage := CONCAT(sMessage, UDINT_TO_STRING(st_Sorter.EncoderCounts));
		// Write to the Error List
		ADSLOGSTR( msgCtrlMask := ADSLOG_MSGTYPE_HINT OR ADSLOG_MSGTYPE_LOG
			, msgFmtStr := CONCAT(st_Sorter.Config.Name, ' Arrival Processed: %s')
			, strArg := sMessage);
	END_IF
	// Indicate that this item did not get added to the sorter and add to the exit buffer
	//  Both as a TransportUpdate and TransportComplete message type 
	IF st_NextToInduct.Item.ID <> '' THEN
		IF nSortBufferLogEnable.BUFFER_MISSINDUCT THEN
			sMessage := CONCAT('Item: ', st_NextToInduct.Item.ID);
			// Write to the Error List
			ADSLOGSTR( msgCtrlMask := ADSLOG_MSGTYPE_HINT OR ADSLOG_MSGTYPE_LOG
				, msgFmtStr := CONCAT(st_Sorter.Config.Name, ' Item Removed - Not Inducted: %s')
				, strArg := sMessage);
		END_IF
		// Transport Response
		st_NextToInduct.Item.Status := E_StatusCode.Assign_NotInducted;
		st_NextToInduct.Item.DeviceID := st_Sorter.Config.EquipID;
		st_NextToInduct.Item.MessageType := E_MessageIds.TransportResponse_25;
		fb_UpdateBuffer.AddItem(st_ItemToAdd := st_NextToInduct.Item);

		// Transport Complete
		st_NextToInduct.Item.Status := E_StatusCode.Divert_NotInducted;
		st_NextToInduct.Item.MessageType := E_MessageIds.TransportComplete_26;
		fb_UpdateBuffer.AddItem(st_ItemToAdd := st_NextToInduct.Item);
	END_IF
	// Copy Last BCR item to Item to Induct
	st_NextToInduct.Item :=  st_ArrivalItem;
	// Add the Sorter EquipID to the NextToInduct
	st_NextToInduct.Item.DeviceID := st_Sorter.Config.EquipID;
	// Set the Default Destination
	IF DestinationOverride = 0 THEN
		st_NextToInduct.Item.Destination := st_Sorter.Config.DefaultDestination;
		st_NextToInduct.Item.DestinationIdx := st_Sorter.Config.DefaultDestIdx;
	ELSE
		st_NextToInduct.Item.Destination := DestinationOverride;
		IF nSorterLogEnable.SORTER_DESTINATION_LU THEN
			sMessage := CONCAT('Destination: ', DINT_TO_STRING(st_NextToInduct.Item.Destination));
			// Write to the Error List
			ADSLOGSTR( msgCtrlMask := ADSLOG_MSGTYPE_HINT OR ADSLOG_MSGTYPE_LOG
				, msgFmtStr := CONCAT(st_sorter.Config.Name, ' Buffer Destination OR Lookup %s')
				, strArg := sMessage);
		END_IF
		fb_FindDestination(RoundRobin := st_Sorter.RoundRobin
						, SorterLogEnable := nSorterLogEnable
						, aDiverts := aTempDiverts
						, DestinationID := st_NextToInduct.Item.Destination
						, DestinationIndex => st_NextToInduct.Item.DestinationIdx);
		
	END_IF
	// Capture an encoder value that when the encoder count exceeds this value, NextToInduct item will be cleared
	st_NextToInduct.Counts := st_Sorter.EncoderCounts;
	// Clear the Last recieved item
	st_ArrivalItem := BlankItem;
	// Prepare to replace the Temporarily assigned item with this item
	IF st_TempInductItem.Item.ID <> '' THEN
		// Capture the Counts and Length from the temporary item
		st_NextToInduct.Counts := st_TempInductItem.Counts;
		st_NextToInduct.Item.Length := st_TempInductItem.Item.Length;
		//Identify the Item to replace in the sorter array
		st_ReplaceItem := st_TempInductItem.Item;
		st_TempInductItem.Counts := 0;
		st_TempInductItem.Item := BlankItem;
		IF nSortBufferLogEnable.BUFFER_TEMPINDUCT THEN
			ADSLOGSTR( msgCtrlMask := ADSLOG_MSGTYPE_HINT OR ADSLOG_MSGTYPE_LOG
				, msgFmtStr := CONCAT(st_Sorter.Config.Name, ' Temp ID Replaced : %s')
				, strArg := st_ReplaceItem.ID); 
		END_IF
	END_IF
END_IF

(*
 	Check for a value disagreement in the SorterTransportBuffer In and Out pointers to
  	determine if there is an update for an item.
	When an update arrived, the System PLC adds it to the shared buffer and increments
	the InPointer
*)
IF st_SorterTransportBufferP6040.nInPointer <> fb_TransportBuffer.OutPointer THEN
	fb_TransportBuffer.RemoveItem(st_ItemToReturn => st_ToUpdate.Item);
	// Override any received destination if there is an Override
	IF DestinationOverride <> 0 THEN
		st_ToUpdate.Item.Destination := DestinationOverride;
	END_IF
	// Lookup the index for the chosen destination
	IF nSorterLogEnable.SORTER_DESTINATION_LU THEN
		sMessage := CONCAT('Destination: ', DINT_TO_STRING(st_ToUpdate.Item.Destination));
		// Write to the Error List
		ADSLOGSTR( msgCtrlMask := ADSLOG_MSGTYPE_HINT OR ADSLOG_MSGTYPE_LOG
			, msgFmtStr := CONCAT(st_sorter.Config.Name, ' Buffer Update Lookup %s')
			, strArg := sMessage);
	END_IF
	fb_FindDestination(RoundRobin := st_Sorter.RoundRobin
					, SorterLogEnable := nSorterLogEnable
					, aDiverts := aTempDiverts
					, DestinationID := st_ToUpdate.Item.Destination
					, DestinationIndex => st_ToUpdate.Item.DestinationIdx);
	IF nSortBufferLogEnable.BUFFER_DESTINDEX THEN
		sMessage := CONCAT('Item: ', st_ToUpdate.Item.ID);
		sMessage := CONCAT(sMessage,' Destination: ');
		sMessage := CONCAT(sMessage, DINT_TO_STRING(st_ToUpdate.Item.Destination));
		sMessage := CONCAT(sMessage,' Index: ');
		sMessage := CONCAT(sMessage, DINT_TO_STRING(st_ToUpdate.Item.DestinationIdx));
		// Write to the Error List
		ADSLOGSTR( msgCtrlMask := ADSLOG_MSGTYPE_HINT OR ADSLOG_MSGTYPE_LOG
			, msgFmtStr := CONCAT(st_Sorter.Config.Name, ' Divert Index of Destination: %s')
			, strArg := sMessage);
	END_IF
END_IF

// Get the Default Destination Index
fb_DefaultDestination(RoundRobin := st_Sorter.RoundRobin
				, NoAssignment := TRUE
				, aDiverts := aTempDiverts
				, DestinationID := st_Sorter.Config.DefaultDestination
				, DestinationIndex => DefaultDestIdx);

// Get the Recirculation Destination Index
fb_RecircDestination(RoundRobin := st_Sorter.RoundRobin
				, NoAssignment := TRUE
				, aDiverts := aTempDiverts
				, DestinationID := st_Sorter.Config.RecircDestination
				, DestinationIndex => RecircDestIdx);

// Test the Item to Update against the Item to Induct and update if they match:
//	Update the NextItemToInduct with the updated data, then clear the Item to Update
IF st_ToUpdate.Item.ID <> '' THEN
	IF st_ToUpdate.Item.ID = st_NextToInduct.Item.ID THEN
		// Indicate that the transport command was received and a response was sent
		st_NextToInduct.Item.MessageType := E_MessageIds.TransportResponse_25;
		// Test the assigned lane for availability
		IF (aDiverts[st_ToUpdate.Item.DestinationIdx].Full
		   OR aDiverts[st_ToUpdate.Item.DestinationIdx].Faulted)
		   AND DestinationOverride = 0
		   THEN
			// Prepare a message to indicate that the item cannot be assigned
			st_ToUpdate.Item.Status := E_StatusCode.Assign_Full;
			st_ToUpdate.Item.DeviceID := st_Sorter.Config.EquipID;
			st_ToUpdate.Item.MessageType := E_MessageIds.TransportResponse_25;
			fb_UpdateBuffer.AddItem(st_ItemToAdd := st_ToUpdate.Item);
			st_NextToInduct.Item.ExtStatus := E_StatusCode.Divert_Full;
		ELSE
			st_NextToInduct.Item.DeviceID := st_Sorter.Config.EquipID;
			st_NextToInduct.Item.Status := E_StatusCode.Assign_Accepted;
			// Update the Destination
			st_NextToInduct.Item.Destination := st_ToUpdate.Item.Destination;
			st_NextToInduct.Item.DestinationIdx := st_ToUpdate.Item.DestinationIdx;
			fb_UpdateBuffer.AddItem(st_ItemToAdd := st_NextToInduct.Item);
		END_IF
		// If commissioning, ignore any other direction
		IF DivertToCommission > 0 THEN
			st_NextToInduct.Item.Destination := DivertToCommission;
		END_IF
		// Log the update
		IF nSortBufferLogEnable.BUFFER_INDUCT THEN
			sMessage := CONCAT('Item: ', st_ToUpdate.Item.ID);
			sMessage := CONCAT(sMessage,' Pulses: ');
			sMessage := CONCAT(sMessage, UDINT_TO_STRING(st_Sorter.EncoderCounts));
			sMessage := CONCAT(sMessage,' Status: ');
			sMessage := CONCAT(sMessage, UDINT_TO_STRING(st_ToUpdate.Item.Status));
			sMessage := CONCAT(sMessage,' Ext Status: ');
			sMessage := CONCAT(sMessage, UDINT_TO_STRING(st_ToUpdate.Item.ExtStatus));
			// Write to the Error List
			ADSLOGSTR( msgCtrlMask := ADSLOG_MSGTYPE_HINT OR ADSLOG_MSGTYPE_LOG
				, msgFmtStr := CONCAT(st_Sorter.Config.Name, ' Found Before Induct: %s')
				, strArg := sMessage);
		END_IF
		// We updated the item we were inducting, clear the Item to update
		st_ToUpdate.Item := BlankItem;
	END_IF
END_IF

// Clear the Update Item Found record each pass
TransportItemFound := BlankItem;

// Clear the last detected Exit item
ExitItemFound.Item := BlankItem;

// Reset the Detection booleans
ExitInDivert := FALSE;
ExitDiverting := FALSE;
ExitDetected := FALSE;
ExitSuccess := FALSE;
ExitComplete := FALSE;

// Loop through the entire array, it should be appropriately sized for the length of the sorter section
FOR UpdateIndexCounter := UDINT_TO_DINT(ItemsArrayMin) TO UDINT_TO_DINT(ItemsArrayMax) DO //Loop through everything in the sorter	

	// For Transport commands, start from the current encoder count and work forwards, just like the exit
	TransportSorterIndex := F_CalculateIndex(Offset := (UpdateIndexCounter)
											, InitialValue := st_Sorter.EncoderCounts
											, BufferSize := ItemsArraySize);

	// This is the item in the sorter array that we will be procesing this pass, testing for a Transport update message
	TransportItemInSorter := aItems[UDINT_TO_DINT(TransportSorterIndex)];

	// Test for a replace item
	// ReplaceItem is the temporary item
	// NextToInduct is the item to replace the temporary with
	IF st_ReplaceItem.ID <> '' THEN
		IF st_ReplaceItem.ID = TransportItemInSorter.ID THEN
			IF nSortBufferLogEnable.BUFFER_REPLACEINDUCT THEN
				sMessage := CONCAT('Item: ', st_ReplaceItem.ID);
				sMessage := CONCAT(sMessage,' New Item: ');
				sMessage := CONCAT(sMessage, st_NextToInduct.Item.ID);
				sMessage := CONCAT(sMessage,' Index: ');
				sMessage := CONCAT(sMessage, UDINT_TO_STRING(TransportSorterIndex));
				sMessage := CONCAT(sMessage,' Orig Dest: ');
				sMessage := CONCAT(sMessage, DINT_TO_STRING(TransportItemInSorter.Destination));
				sMessage := CONCAT(sMessage,' New Dest: ');
				sMessage := CONCAT(sMEssage, DINT_TO_STRING(st_ReplaceItem.Destination));
				sMessage := CONCAT(sMessage,' Orig Idx: ');
				sMessage := CONCAT(sMessage, DINT_TO_STRING(TransportItemInSorter.DestinationIdx));
				sMessage := CONCAT(sMessage,' New Idx: ');
				sMessage := CONCAT(sMEssage, DINT_TO_STRING(st_ReplaceItem.DestinationIdx));
				// Write to the Error List
				ADSLOGSTR( msgCtrlMask := ADSLOG_MSGTYPE_HINT OR ADSLOG_MSGTYPE_LOG
					, msgFmtStr := CONCAT(st_Sorter.Config.Name, ' Item ID Replaced After Induct: %s')
					, strArg := sMessage);
			END_IF
			TransportItemInSorter.ID := st_NextToInduct.Item.ID;
			TransportItemInSorter.Destination := st_NextToInduct.Item.Destination;
			TransportItemInSorter.DestinationIdx := st_NextToInduct.Item.DestinationIdx;
			TransportItemInSorter.DeviceID := st_NextToInduct.Item.DeviceID;
			TransportItemInSorter.MessageType := st_NextToInduct.Item.MessageType;
			TransportItemInSorter.Status := st_NextToInduct.Item.Status;
			TransportItemInSorter.UniqueID := st_NextToInduct.Item.UniqueID;
			TransportItemInSorter.CapturedInMetrics := st_NextToInduct.Item.CapturedInMetrics;
		END_IF
	END_IF
	// Test for an Item Update
	IF st_ToUpdate.Item.ID <> '' THEN
		// Test the sorter item against the update item
		IF st_ToUpdate.Item.ID = TransportItemInSorter.ID THEN
			IF nSortBufferLogEnable.BUFFER_UPDATEINDUCT THEN
				sMessage := CONCAT('Item: ', st_ToUpdate.Item.ID);
				sMessage := CONCAT(sMessage,' Index: ');
				sMessage := CONCAT(sMessage, UDINT_TO_STRING(TransportSorterIndex));
				// Write to the Error List
				ADSLOGSTR( msgCtrlMask := ADSLOG_MSGTYPE_HINT OR ADSLOG_MSGTYPE_LOG
					, msgFmtStr := CONCAT(st_Sorter.Config.Name, ' Found After Induct: %s')
					, strArg := sMessage);
			END_IF
			// Copy the found item record, 
			TransportItemFound := TransportItemInSorter;
			// Test the destined divert for availability
			IF aDiverts[st_ToUpdate.Item.DestinationIdx].Full OR aDiverts[st_ToUpdate.Item.DestinationIdx].Faulted THEN
				// Prepare a message to indicate that the item cannot be assigned
				TransportItemFound.Status := E_StatusCode.Assign_Full;
				TransportItemFound.ExtStatus := E_StatusCode.Divert_Full;
				TransportItemFound.MessageType := E_MessageIds.TransportResponse_25;
				TransportItemFound.Destination := st_Sorter.Config.DefaultDestination;
				TransportItemFound.DestinationIdx := st_Sorter.Config.DefaultDestIdx;
			// Test for an already diverting item and assign an ExtStatus of LateAssignment
			ELSIF TransportItemInSorter.Status >= E_StatusCode.Diverting THEN
				TransportItemFound.ExtStatus := E_StatusCode.Divert_LateAssignment;
				TransportItemFound.MessageType := E_MessageIds.TransportResponse_25;
			ELSE
				//  Change the destination, which should be the only item in the update
				TransportItemFound.Destination := st_ToUpdate.Item.Destination;
				TransportItemFound.DestinationIdx := st_ToUpdate.Item.DestinationIdx;
				// This message indicates we could assign the Item
				TransportItemFound.Status := E_StatusCode.Assign_Accepted;
				TransportItemFound.MessageType := E_MessageIds.TransportResponse_25;
			END_IF
			TransportItemFound.DeviceID := st_Sorter.Config.EquipID;
			// Add the item to the update buffer
			fb_UpdateBuffer.AddItem(TransportItemFound);
			// Clear the ToUpdate Item
			st_ToUpdate.Item := BlankItem;
		END_IF
	END_IF
	
	IF TransportItemFound.ID <> '' THEN
		// Test the sorter item against the update item
		IF TransportItemFound.ID = TransportItemInSorter.ID THEN
			// Only update if it is different
			IF TransportItemFound.Destination <> TransportItemInSorter.Destination THEN
				IF nSortBufferLogEnable.BUFFER_UPDATEDEST THEN
					sMessage := CONCAT('Item: ', TransportItemInSorter.ID);
					sMessage := CONCAT(sMessage,' Index: ');
					sMessage := CONCAT(sMessage, UDINT_TO_STRING(TransportSorterIndex));
					sMessage := CONCAT(sMessage,' Orig Dest: ');
					sMessage := CONCAT(sMessage, DINT_TO_STRING(TransportItemInSorter.Destination));
					sMessage := CONCAT(sMessage,' Orig Idx: ');
					sMessage := CONCAT(sMessage, DINT_TO_STRING(TransportItemInSorter.DestinationIdx));
					sMessage := CONCAT(sMessage,' Orig DeviceID ');
					sMessage := CONCAT(sMessage, TransportItemInSorter.DeviceID);
					// Write to the Error List
					ADSLOGSTR( msgCtrlMask := ADSLOG_MSGTYPE_HINT OR ADSLOG_MSGTYPE_LOG
						, msgFmtStr := CONCAT(st_Sorter.Config.Name, ' Dest Updated After Induct: %s')
						, strArg := sMessage);
				END_IF
				// Update the Destination. If the destination is unavailable, it has been already been set to the default
				TransportItemInSorter.Destination := TransportItemFound.Destination;
				TransportItemInSorter.DestinationIdx := TransportItemFound.DestinationIdx;
				TransportItemInSorter.DeviceID := TransportItemFound.DeviceID;
				TransportItemInSorter.MessageType := TransportItemFound.MessageType;
				TransportItemInSorter.Status := TransportItemFound.Status;
				TransportItemInSorter.ExtStatus := TransportItemFound.ExtStatus;
	
